IF bMove THEN
    CASE eHomeState OF
        // Wait for a rising edge
        E_MoveState.IDLING:
            IF bHomeModeEnabled AND bExecHome THEN
                bHomeDone := FALSE;
                bHomeBusy := TRUE;
                stMotionStage.bDone := FALSE;
                stDS402Drive.nDriveControl:=15;
                eHomeState :=  E_MoveState.INIT;
            END_IF
        E_MoveState.INIT:
                        stDS402Drive.nDriveControl.4:=1;
                                        eHomeState := E_MoveState.STARTED;
        E_MoveState.STARTED :
            // this is a comfirmation that routine is ongoing
            IF NOT stDS402Drive.stDriveStatus.TargetReached
                AND NOT stDS402Drive.stDriveStatus.Bit13_OpModeSpecific THEN
                bHomeBusy:=TRUE;
                bHomeDone:=FALSE;

                eHomeState:=E_MoveState.IN_PROGRESS;
            END_IF

        E_MoveState.IN_PROGRESS :

        IF bStop THEN
         stDS402Drive.nDriveControl.8 :=1;
          bHomeAborted := TRUE;
          eHomeState:=E_MoveState.INTERRUPTED;

        // Genral Motion error i.e Following error ?
        ELSIF stDS402Drive.stDriveStatus.Bit13_OpModeSpecific
                OR stDS402Drive.stDriveStatus.WarningCondition THEN
            stMotionStage.bError := TRUE;
            eHomeState:=E_MoveState.ERROR;

        // Reached
        ELSIF stDS402Drive.stDriveStatus.TargetReached
            AND stDS402Drive.stDriveStatus.Bit12_OpModeSpecific
            AND NOT stDS402Drive.stDriveStatus.Bit13_OpModeSpecific THEN
           eHomeState:=E_MoveState.DONE;
        END_IF
        E_MoveState.INTERRUPTED:
            bHomeBusy:=FALSE;
            eHomeState:=E_MoveState.IDLING;
        E_MoveState.DONE:
            bHomeBusy:=FALSE;
            bHomeDone:=TRUE;
            stMotionStage.fPosition:=0.0;

            IF (stMotionStage.nEnableMode = E_StageEnableMode.DURING_MOTION ) THEN
                stDS402Drive.nDriveControl.4:=FALSE;

            ELSE
                stDS402Drive.nDriveControl:=6;
            END_IF
            eHomeState:=E_MoveState.IDLING;
        E_MoveState.ERROR:
            bHomeDone:=FALSE;
            bHomeBusy:= FALSE;
            IF bWrongParameter THEN
                stMotionStage.sCustomErrorMessage:='Invalid motion Parameters';
                bWrongParameter := FALSE;
                stMotionStage.bError := TRUE;
            END_IF
            IF NOT stMotionStage.bError THEN
                eHomeState:=E_MoveState.IDLING;
            END_IF
    END_CASE
END_IF
END_METHOD

METHOD PUBLIC Interlock

VAR_INST
    {attribute 'hide'}
    bPositiveDirection  : BOOL;
    {attribute 'hide'}
    bNegativeDirection  : BOOL;
    {attribute 'hide'}
    ftForwardEnabled  	: F_TRIG;

    {attribute 'hide'}
    ftBackwardEnabled 	: F_TRIG;
END_VAR
// Positive or Negative direction
bPositiveDirection:=stMotionStage.bBusy AND stMotionStage.fPosDiff > 0;
bNegativeDirection:=stMotionStage.bBusy AND stMotionStage.fPosDiff < 0;

// For SmartAct MCS2 these limit are range and enstop limits. however a single bit in the status is used
// bLimOverride  : act as an override after limit was hit to allow reverse movement
stMotionStage.bLimitForwardEnable :=  bLimOverride OR NOT( bPositiveDirection AND stDS402Drive.stDriveStatus.InternalLimitActive );
stMotionStage.bLimitBackwardEnable := bLimOverride OR NOT( bNegativeDirection AND stDS402Drive.stDriveStatus.InternalLimitActive );

// use falling trigger to avoid spaming  sErrorMessage
ftForwardEnabled(CLK:=stMotionStage.bLimitForwardEnable);
ftBackwardEnabled(CLK:=stMotionStage.bLimitBackwardEnable);

IF  NOT bHomeBusy AND ftForwardEnabled.Q THEN
    // Not an error, just a warning
    stMotionStage.sCustomErrorMessage:='Cannot move past positive limit.';
    bLimOverride := TRUE;
END_IF

IF NOT bHomeBusy AND ftBackwardEnabled.Q THEN
    // Not an error, just a warning
    stMotionStage.sCustomErrorMessage:='Cannot move past Negative limit.';
    bLimOverride := TRUE;
END_IF

IF NOT stMotionStage.bError AND stMotionStage.bExecute AND NOT stMotionStage.bUserEnable THEN
    stMotionStage.bError := TRUE;
    stMotionStage.nErrorId := 1;
    stMotionStage.sCustomErrorMessage := 'Move requested, but user enable is disabled!';
END_IF

// Update all enable booleans
SetEnables();
END_METHOD

(*Switch the drive mod eof Operation
  Servo On: Profil Positioning or HOME
  Servo Off : STEP mode
*)
METHOD ModeOperation

VAR_INST
    tonSwitching : TON;
    bManualTransition: BOOL;
END_VAR
rtCSPModeOk(CLK:=( stDS402Drive.nModeOfOperationDisplay=E_DS402OpMode.CSP));
rtHomeModeEnable(CLK:=( stDS402Drive.nModeOfOperationDisplay=E_DS402OpMode.HOME));
// transition to close loop mode
IF rtCSPModeOk.Q THEN
    bHomeModeEnabled := FALSE;
    bCSPModeEnabled := TRUE;
ELSIF rtHomeModeEnable.Q THEN
    bHomeModeEnabled := TRUE;
    bCSPModeEnabled := FALSE;
    stDS402Drive.nDriveControl := 0;
END_IF

IF rtUserExec.Q AND stMotionStage.bHomeCmd THEN
    IF (stDS402Drive.nModeOfOperationDisplay<>E_DS402OpMode.HOME) THEN
        stDS402Drive.nModeOfOperation := E_DS402OpMode.HOME;
        stDS402Drive.nDriveControl := 128;
        // clear previous operational from switching away from this mode.
        bOperational := FALSE;
        bCSPModeEnabled := FALSE;
        bManualTransition := TRUE;
    ELSE
        bHomeModeEnabled := TRUE;
    END_IF
ELSIF rtUserExec.Q THEN
    IF (stDS402Drive.nModeOfOperationDisplay<>E_DS402OpMode.CSP) THEN
        stDS402Drive.nModeOfOperation := E_DS402OpMode.CSP;
        stDS402Drive.nDriveControl := 128;
        bHomeModeEnabled := FALSE;
        bManualTransition := FALSE;
    ELSE
        bCSPModeEnabled := TRUE;
    END_IF
END_IF

bDS402ManualEnabled :=bHomeModeEnabled;
(*Handle correct startup procedure for manual move*)
StateMachine(Enable:=1);
END_METHOD

METHOD PUBLIC  MoveAbsolute

fbMcMoveAbsolute(
    Axis := stMotionStage.Axis,
    Execute := bCommandMoveAbsolute,
    Position := stMotionStage.fPosition,
    Velocity := stMotionStage.fVelocity,
    Acceleration := stMotionStage.fAcceleration,
    Deceleration := stMotionStage.fDeceleration,
    BufferMode := eBufferMode,
);
END_METHOD

METHOD PersistParameters
VAR_INPUT
    Enable	: BOOL;
END_VAR

VAR_INST
    {attribute 'hide'}
    bEncError			: BOOL;

    {attribute 'hide'}
    bRestoreWaitRetry	: BOOL;
END_VAR
// Save Encoder position
// needs some pre-conditions to use persistent storage
IF Enable THEN
    // Check ST_MotionStage for an encoder error (range 0x44nn)
    bEncError:= stMotionStage.Axis.Status.Error AND  ( stMotionStage.Axis.Status.ErrorID  >= 16#4400  AND stMotionStage.Axis.Status.ErrorID <= 16#44FF );
    // Do not save if we're currently loading or if there is an encoder error
    IF NOT bRestoreLoad AND NOT bEncError AND NOT bRestoreWaitRetry THEN
        fSavedPosition := stMotionStage.Axis.NcToPlc.ActPos;
        // This persistent variable lets us check if anything was saved
        // It will be TRUE at startup if we have saved values
        bSaved := TRUE;
        (*
            use this with a timer of a change threshold on the fActPosition
            to trigger a save from this PLC program. otherwise this will be a spamming
            persistence, filling up the disk.
        *)
        //iPersistentDataStorage.TriggerWriteOfPersistentData := bSaveEnabled;
    END_IF
END_IF
END_METHOD

{attribute 'call_after_init'}
(*	eModule: Mandatory must be unique for each MCS2 axis
    clears startup errors or warnings. the process is completed at run time
    SDO update of Drive and open Loop parameter Indexes based on module number
*)
METHOD PostInit
VAR_INPUT
END_VAR
(* SDO update of Drive and open Loop parameter Indexes based on module number*)
nChanErrorCodeIdx	:= nErrorCodeBase		+ ((eModule-1) * nChanOfsBase);
nChanSoftLimitIdx	:= nChanSoftLimitBase 	+ ((eModule-1) * nChanOfsBase);
bInit := TRUE;
END_METHOD

METHOD Power : BOOL
fbMcPower(
    Axis := stMotionStage.Axis,
    Enable := stMotionStage.bAllEnable AND bCSPModeEnabled,
    Enable_Positive := stMotionStage.bAllForwardEnable,
    Enable_Negative := stMotionStage.bAllBackwardEnable,
    Override := 100.0,
    BufferMode := eBufferMode );
END_METHOD

(* Read Drive error codes after a motion or fault condition occured *)
METHOD ReadDriveCodes : BOOL
VAR_INST
    {attribute 'hide'}
    fbErrorRead			: FB_EcCoESdoRead;
    {attribute 'hide'}
    nPiezoErrorCode   	: UDINT;
    {attribute 'hide'}
    fbLogError  		: FB_LogMotionError;
    {attribute 'hide'}
    ftErrorReadDone  	: F_TRIG;
END_VAR
fbErrorRead( sNetId:= THIS^.stMotionStage.stAxisParameters.sAmsNetId,
             nSlaveAddr:=stDS402Drive.nSlaveAddr,
             nIndex:=nChanErrorCodeIdx,
             nSubIndex :=nSubIndex,
             pDstBuf:= ADR(nPiezoErrorCode),
             cbBufLen:=SIZEOF(nPiezoErrorCode),
             bExecute:= stMotionStage.bError );

ftErrorReadDone(CLK:=fbErrorRead.bBusy);
IF ftErrorReadDone.Q THEN
    IF 	NOT fbErrorRead.bError AND nPiezoErrorCode <> 0 THEN
        stMotionStage.nErrorId := nPiezoErrorCode;
    END_IF
    stMotionStage.sErrorMessage := F_MotionErrorCodeLookup(nErrorId:=stMotionStage.nErrorId);
    fbLogError( stMotionStage:=stMotionStage, bEnable:=stMotionStage.bError);
END_IF
END_METHOD

METHOD Reset : BOOL
fbMcReset(
    Axis := stMotionStage.Axis,
    Execute := bLocalReset AND bCSPModeEnabled
);

IF fbMcReset.Done OR fbMcReset.Error THEN
    bLocalReset := FALSE;
END_IF
END_METHOD

METHOD RestoreMotionParams
VAR_INPUT
    Enable	: BOOL;
END_VAR

VAR_INST
    {attribute 'hide'}
    fbSetPos			: MC_SetPosition;
    {attribute 'hide'}
    bLoad				: BOOL;
    {attribute 'hide'}
    bRestoreDone 		: BOOL;
    {attribute 'hide'}
    bRestoreInit		: BOOL;
    {attribute 'hide'}
    bRestoreWaitRetry	: BOOL;
    {attribute 'hide'}
    nMaxRetries			: UINT := 10;
    {attribute 'hide'}
    nCurrTries			: UINT := 0;
    {attribute 'hide'}
    nLatchError			: UDINT;
END_VAR
IF Enable THEN
    // Trigger a load if anything was saved at all
    IF NOT bRestoreInit THEN
        bRestoreInit := TRUE;
        bRestoreLoad S= bSaved;
        fbSetPos.Options.ClearPositionLag := TRUE;
    END_IF

    // Set our position if bRestoreLoad is true
    fbSetPos( Axis:=stMotionStage.Axis, Execute:=bRestoreLoad, Position:=fSavedPosition);

    // Only load once, at startup
    bRestoreLoad R= fbSetPos.Done OR fbSetPos.Error;

    IF fbSetPos.Error THEN
        // Keep the error latched, it can disappear if Execute is set to FALSE
        nLatchError := fbSetPos.ErrorID;
        nCurrTries := nCurrTries + 1;
        IF nCurrTries >= nMaxRetries THEN
        // Alert the user that something has gone wrong
        stMotionStage.bError := TRUE;
        stMotionStage.nErrorId := nLatchError;
        stMotionStage.sCustomErrorMessage := 'Error loading previously saved position.';
        ELSE
            // Reset the FB for the next retry
            fbSetPos( Axis:=stMotionStage.Axis, Execute:=bRestoreLoad, Position:=fSavedPosition);
            // Try again
            bRestoreWaitRetry := TRUE;
        END_IF
    ELSE
        IF NOT bRestoreDone THEN
            stMotionStage.fPosition := fSavedPosition;
        END_IF
        bRestoreDone := TRUE;
    END_IF

    tonRestoreRetry( IN := bRestoreWaitRetry, PT := T#100MS);
    bRestoreLoad S= tonRestoreRetry.Q;
    bRestoreWaitRetry R= tonRestoreRetry.Q;
END_IF
END_METHOD

METHOD ScaleDriveParams
nSoftLimMax := LREAL_TO_DINT((stMotionStage.stAxisParameters.fEncSoftEndMax / MAX(stMotionStage.stAxisParameters.fEncScaleFactorInternal, fScalingFactor)));
nSoftLimMin := LREAL_TO_DINT((stMotionStage.stAxisParameters.fEncSoftEndMin / MAX(stMotionStage.stAxisParameters.fEncScaleFactorInternal, fScalingFactor)));
END_METHOD

METHOD ScaleEncRawValue
VAR_INPUT
  //  bEnable: BOOL;
END_VAR
(* SmartACT: The encoder count from the Piezo drive is not a raw count from the embeded actuator device
   we get a calibrated nm value. thus the use of abs() since this value is signed.
   PI: to be discovered *)
IF stMotionStage.nRawEncoderDINT <> 0 THEN
    stMotionStage.nEncoderCount:=DINT_TO_UDINT(ABS(stMotionStage.nRawEncoderDINT));
ELSE
    stMotionStage.nEncoderCount:=0;
END_IF

// calibrated encoder readback
fMeasuredPos:=stMotionStage.Axis.NcToPlc.ActPos;
fMeasuredVelo :=stMotionStage.Axis.NcToPlc.ActVelo;
fMeasuredAcc := stMotionStage.Axis.NcToPlc.ActAcc;
stMotionStage.fPosDiff:=stMotionStage.Axis.NcToPlc.PosDiff;
END_METHOD

METHOD SetEnables
VAR_INPUT
END_VAR
stMotionStage.bAllForwardEnable:=stMotionStage.bLimitForwardEnable AND (stMotionStage.bGantryForwardEnable OR NOT stMotionStage.bGantryAxis) AND stMotionStage.stEPSForwardEnable.bEPS_OK;
stMotionStage.bAllBackwardEnable:=stMotionStage.bLimitBackwardEnable AND (stMotionStage.bGantryBackwardEnable OR NOT stMotionStage.bGantryAxis) AND stMotionStage.stEPSBackwardEnable.bEPS_OK;

stMotionStage.bAllEnable:=stMotionStage.bEnable AND stMotionStage.bHardwareEnable AND stMotionStage.stEPSPowerEnable.bEPS_OK;
stMotionStage.bAllEnable R= NOT stMotionStage.bUserEnable;
END_METHOD

METHOD StateMachine
VAR_INPUT
    Enable : BOOL;
END_VAR

VAR_INST
    rtFault: R_TRIG;
    {attribute 'hide'}
    bFault				: BOOL;
END_VAR
rtFault(CLK:=bFault);
(*switch on disable*)
IF NOT stDS402Drive.stDriveStatus.ReadyToSwitchOn
    AND NOT stDS402Drive.stDriveStatus.SwitchedOn
    AND NOT stDS402Drive.stDriveStatus.OperationEnabled
    AND NOT stDS402Drive.stDriveStatus.Fault
    AND stDS402Drive.stDriveStatus.VoltageEnabled
    AND NOT stDS402Drive.stDriveStatus.QuickStopActive
    AND  stDS402Drive.stDriveStatus.SwitchOnDisabled THEN
        bOperational := FALSE;
        IF bDS402ManualEnabled AND NOT bStop  THEN
            THIS^.stDS402Drive.nDriveControl := 6;
        END_IF
(*Ready to switch*)
ELSIF stDS402Drive.stDriveStatus.ReadyToSwitchOn
    AND NOT stDS402Drive.stDriveStatus.SwitchedOn
    AND NOT stDS402Drive.stDriveStatus.OperationEnabled
    AND NOT stDS402Drive.stDriveStatus.Fault
    AND stDS402Drive.stDriveStatus.VoltageEnabled
    AND stDS402Drive.stDriveStatus.QuickStopActive
    AND NOT stDS402Drive.stDriveStatus.SwitchOnDisabled THEN
        bFault := FALSE;
        bOperational := FALSE;
        IF bDS402ManualEnabled AND NOT bStop  THEN
            THIS^.stDS402Drive.nDriveControl := 7;
        END_IF
(*Switch on*)
ELSIF stDS402Drive.stDriveStatus.ReadyToSwitchOn
    AND  stDS402Drive.stDriveStatus.SwitchedOn
    AND NOT stDS402Drive.stDriveStatus.OperationEnabled
    AND NOT stDS402Drive.stDriveStatus.Fault
    AND stDS402Drive.stDriveStatus.VoltageEnabled
    AND stDS402Drive.stDriveStatus.QuickStopActive
    AND NOT stDS402Drive.stDriveStatus.SwitchOnDisabled THEN
        bOperational := FALSE;
        IF bDS402ManualEnabled AND NOT bStop  THEN
            THIS^.stDS402Drive.nDriveControl := 15;
        END_IF
(*Operation enbaled*)
ELSIF stDS402Drive.stDriveStatus.ReadyToSwitchOn
    AND stDS402Drive.stDriveStatus.SwitchedOn
    AND stDS402Drive.stDriveStatus.OperationEnabled
    AND NOT stDS402Drive.stDriveStatus.Fault
    AND stDS402Drive.stDriveStatus.VoltageEnabled
    AND stDS402Drive.stDriveStatus.QuickStopActive
    AND NOT stDS402Drive.stDriveStatus.SwitchOnDisabled THEN
        THIS^.bOperational := TRUE;
(*Fault*)
ELSIF  NOT stDS402Drive.stDriveStatus.ReadyToSwitchOn
    AND NOT stDS402Drive.stDriveStatus.SwitchedOn
    AND NOT stDS402Drive.stDriveStatus.OperationEnabled
    AND stDS402Drive.stDriveStatus.Fault
    AND stDS402Drive.stDriveStatus.VoltageEnabled
    AND NOT stDS402Drive.stDriveStatus.QuickStopActive
    AND NOT stDS402Drive.stDriveStatus.SwitchOnDisabled THEN
        bOperational := FALSE;
        bFault := TRUE;

ELSE
    bFault := FALSE;
    bOperational := FALSE;
END_IF

// wait for parameter init done at startup to read potential error from drive
stMotionStage.bError := bFault AND stMotionStage.bAxisParamsInit;
END_METHOD

(*	Drive parameters update
    Mirror NC axis parameters configurations to those of MCS2 drive
    1- Following error
    2- Home Speeds
    3- Home Acceleration
    4- SoftLimits
*)
METHOD UpdateDriveMonitoringParams
VAR_INPUT
    Enable : BOOL;
END_VAR

VAR_INST
    {attribute 'hide'}
    fbSetFErrorWin		: FB_EcCoESdoWrite;
    {attribute 'hide'}
    fbSetSoftLimMin		: FB_EcCoESdoWrite;
    {attribute 'hide'}
    fbSetSoftLimMax		: FB_EcCoESdoWrite;
    {attribute 'hide'}
    fbSetHomeOffs 		: FB_EcCoESdoWrite;
    {attribute 'hide'}
    fbSetHomeVeloFast 	: FB_EcCoESdoWrite;
    {attribute 'hide'}
    fbSetHomeVeloSlow 	: FB_EcCoESdoWrite;
    {attribute 'hide'}
    fbSetHomeAcc		: FB_EcCoESdoWrite;
    {attribute 'hide'}
    nRecentSoftLimMax 	: LINT;
    {attribute 'hide'}
    nRecentSoftLimMin 	: LINT;
    {attribute 'hide'}
    nRecentHomeVeloFast : UDINT;
    {attribute 'hide'}
    nRecentHomeVeloSlow : UDINT;
    {attribute 'hide'}
    nRecentHomeAcc 		: UDINT;
    {attribute 'hide'}
    nRecentFErrWin		: DINT;
    {attribute 'hide'}
    nRecentHomeOffset 	: DINT;
    {attribute 'hide'}
    nHomeOffs			: DINT;
    {attribute 'hide'}
    ftFErrWinSetDone	: F_TRIG;

    {attribute 'hide'}
    ftSoftLimMaxSetDone	: F_TRIG;
    {attribute 'hide'}
    ftSoftLimMinSetDone	: F_TRIG;
    {attribute 'hide'}
    ftHomeVeloFastSetDone: F_TRIG;
    {attribute 'hide'}
    ftHomeAccSetDone	: F_TRIG;
    {attribute 'hide'}
    ftHomeOffsSetDone	: F_TRIG;
    {attribute 'hide'}
    ftHomeVeloSlowSetDone: F_TRIG;
END_VAR
IF Enable THEN

    (*	Drive parameters update
        Mirror NC axis parameters configurations to those of MCS2 drive
        1- Following error.
        2- SoftLimits
        3-Position Range
    *)
  // add some safety here for  0 div.
  ScaleDriveParams();

  fbSetSoftLimMin(
    sNetId     := THIS^.stMotionStage.stAxisParameters.sAmsNetId,
    nSlaveAddr := stDS402Drive.nSlaveAddr,
    nIndex     := nChanSoftLimitIdx,
    nSubIndex  := 1,
    pSrcBuf    := ADR(nSoftLimMin),
    cbBufLen   := SIZEOF(nSoftLimMin),
    bExecute   := NOT stMotionStage.bBusy AND (nSoftLimMin <> nRecentSoftLimMin)
  );
  fbSetSoftLimMax(
    sNetId     := THIS^.stMotionStage.stAxisParameters.sAmsNetId,
    nSlaveAddr := stDS402Drive.nSlaveAddr,
    nIndex     := nChanSoftLimitIdx,
    nSubIndex  := 2,
    pSrcBuf    := ADR(nSoftLimMax),
    cbBufLen   := SIZEOF(nSoftLimMax),
    bExecute   := NOT stMotionStage.bBusy AND (nSoftLimMax <> nRecentSoftLimMax)
    );

  ftSoftLimMaxSetDone(CLK:=fbSetSoftLimMax.bBusy);
  ftSoftLimMinSetDone(CLK:=fbSetSoftLimMin.bBusy);

    IF ftSoftLimMaxSetDone.Q OR ftSoftLimMinSetDone.Q  THEN
        IF fbSetSoftLimMin.bError THEN
           stMotionStage.bError := fbSetSoftLimMin.bError;
           stMotionStage.nErrorId := fbSetSoftLimMin.nErrId;
        ELSIF fbSetSoftLimMax.bError THEN
           stMotionStage.bError := fbSetSoftLimMax.bError;
           stMotionStage.nErrorId := fbSetSoftLimMax.nErrId;
        ELSE
           nRecentSoftLimMax := nSoftLimMax;
           nRecentSoftLimMin := nSoftLimMin;
        END_IF
        fbSetSoftLimMin.bExecute := FALSE;
        fbSetSoftLimMax.bExecute := FALSE;
    END_IF
END_IF
END_METHOD

METHOD UpdateEpicsStatus
VAR_INPUT
END_VAR
//////////////////////////////////////////////////////////////////
// Transfer NC parameter status to EPICS
//////////////////////////////////////////////////////////////////
stMotionStage.stAxisStatus.bEnable:=stMotionStage.bAllEnable;
stMotionStage.stAxisStatus.bEnabled:=stMotionStage.bEnableDone; // account for PowerEnable from power block
stMotionStage.stAxisStatus.bError:=stMotionStage.bError;
stMotionStage.stAxisStatus.bHomeSensor:=stMotionStage.bHome;
stMotionStage.stAxisStatus.bLimitBwd:=stMotionStage.bAllBackwardEnable;
stMotionStage.stAxisStatus.bLimitFwd:=stMotionStage.bAllForwardEnable;
stMotionStage.stAxisStatus.bReset:=stMotionStage.bReset;
stMotionStage.stAxisStatus.fAcceleration:=fMeasuredAcc;
stMotionStage.stAxisStatus.fActDiff:=stMotionStage.fPosDiff;
stMotionStage.stAxisStatus.fActPosition:=fMeasuredPos;
stMotionStage.stAxisStatus.fActVelocity:=fMeasuredVelo;
stMotionStage.stAxisStatus.fDeceleration:=fMeasuredAcc;
stMotionStage.stAxisStatus.fOverride:=THIS^.fbMcPower.Override;
stMotionStage.stAxisStatus.fPosition:=stMotionStage.fPosition;
stMotionStage.stAxisStatus.fVelocity:=stMotionStage.fVelocity;
stMotionStage.stAxisStatus.nCmdData:=INT_TO_UINT(stMotionStage.nCmdData);  //Or nCmdDataLocal
stMotionStage.stAxisStatus.nCommand:=INT_TO_UINT(stMotionStage.nCommand);  //Or nCommandLocal
stMotionStage.stAxisStatus.nErrorId:=stMotionStage.nErrorId;
stMotionStage.stAxisStatus.bBusy:=stMotionStage.bBusy;
stMotionStage.stAxisStatus.bHomed:=stMotionStage.bHomed;
stMotionStage.stAxisStatus.bExecute:=bLocalExec;
stMotionStage.stAxisStatus.nCommand:=3; // If this is not 3, the IOC stops updating positions during homing
END_METHOD

METHOD WriteParameterNC
VAR_INPUT
    Execute:BOOL;
    ParameterNumber : MC_AxisParameter;
    ParameterValue	: LREAL;
END_VAR
(*Do not change a moving axis parameter*)
fbMcWriteParameter(	Axis:=stMotionStage.Axis,
                    Execute:=(Execute AND stMotionStage.Axis.Status.NotMoving),
                    ParameterNumber:=ParameterNumber,
                    Value:=ParameterValue
                  );

// Reset execute after when done successfull or after abort reset
// this way the done and error condition is latched till next move or global reset.
END_METHOD

END_FUNCTION_BLOCK

// ---- POUs/Motion/DS402/MCS2/FB_MCS2Calibrate.TcPOU
FUNCTION_BLOCK FB_MCS2Calibrate
VAR_INPUT
    bExecute : BOOL;
END_VAR
VAR_IN_OUT
    stDS402Drive         : ST_DS402Drive;
    stMotionStage        : ST_MotionStage;
END_VAR

VAR_OUTPUT
    bCalibrateMoveBusy        : BOOL;
    bCalibrateMoveDone        : BOOL;
    bCalibrateMoveAborted     : BOOL;
END_VAR
VAR
    eStepState	: E_MoveState := E_MoveState.IDLING;
    {attribute 'hide'}
    bReset :  BOOL;
    {attribute 'hide'}
    bHalt : BOOL;
    {attribute 'hide'}
    tonSettlingTime     : TON;
    {attribute 'hide'}
    rtCalibrateMove: R_TRIG;
END_VAR

IF NOT __ISVALIDREF(stDS402Drive)
    OR NOT __ISVALIDREF(stMotionStage) THEN
   RETURN;
END_IF

rtCalibrateMove(CLK := bExecute);

CASE eStepState OF

    E_MoveState.IDLING:
        IF rtCalibrateMove.Q THEN
            bCalibrateMoveBusy := TRUE;
            bCalibrateMoveDone := FALSE;
            // Set bits 0-3 for calibration enable
            stDS402Drive.nDriveControl.3 := TRUE;
            eStepState := E_MoveState.INIT;
        END_IF

    E_MoveState.INIT:
        // Always run the routine, even when the drive reports Calibration Attained
        // (Bit12): a Safe-Direction change invalidates the stored calibration while
        // leaving Bit12 set, so re-calibration must not be skipped.
        IF stMotionStage.bError THEN
            eStepState := E_MoveState.ERROR;
        ELSE
            stDS402Drive.nDriveControl.4 := TRUE;
            tonSettlingTime.IN:=TRUE;
            eStepState := E_MoveState.IN_PROGRESS;
        END_IF

    E_MoveState.IN_PROGRESS:
        IF bHalt OR bReset THEN
            bCalibrateMoveAborted := TRUE;
            eStepState := E_MoveState.INTERRUPTED;
        ELSIF stDS402Drive.stDriveStatus.Bit13_OpModeSpecific THEN
            stMotionStage.bError := TRUE;
            eStepState := E_MoveState.ERROR;
        ELSE
            IF tonSettlingTime.Q AND stDS402Drive.stDriveStatus.TargetReached
              AND stDS402Drive.stDriveStatus.Bit12_OpModeSpecific THEN
                eStepState := E_MoveState.REACHED;
            END_IF
        END_IF

    E_MoveState.INTERRUPTED:
        stDS402Drive.nDriveControl.4 := FALSE;
        bCalibrateMoveBusy := FALSE;
        eStepState := E_MoveState.IDLING;

    E_MoveState.REACHED:
        bCalibrateMoveBusy := FALSE;
        bCalibrateMoveDone := TRUE;
        stDS402Drive.nDriveControl.4 := FALSE;
        eStepState := E_MoveState.DONE;
    E_MoveState.DONE:
        IF stMotionStage.bDone THEN
            eStepState := E_MoveState.IDLING;
        END_IF
    E_MoveState.ERROR:
        bCalibrateMoveBusy := FALSE;
        IF NOT stMotionStage.bError THEN
            eStepState := E_MoveState.IDLING;
        END_IF

END_CASE

tonSettlingTime(PT:=T#80MS);
bHalt := FALSE;
bReset := FALSE;

METHOD Halt : BOOL
VAR_INPUT
END_VAR
THIS^.bHalt := TRUE;
END_METHOD

METHOD Reset : BOOL
VAR_INPUT
END_VAR
THIS^.bReset := TRUE;
END_METHOD

END_FUNCTION_BLOCK

// ---- POUs/Motion/DS402/MCS2/FB_MCS2Home.TcPOU
FUNCTION_BLOCK FB_MCS2Home
VAR_INPUT
    bExecute : BOOL;
END_VAR
VAR_IN_OUT
    stDS402Drive         : ST_DS402Drive;
    stMotionStage        : ST_MotionStage;
END_VAR

VAR_OUTPUT
    bHomeMoveBusy        : BOOL;
    bHomeMoveDone        : BOOL;
    bHomeMoveAborted     : BOOL;
END_VAR
VAR
    eStepState           : E_MoveState := E_MoveState.IDLING;
    {attribute 'hide'}
    bReset :  BOOL;
    {attribute 'hide'}
    bHalt : BOOL;
    {attribute 'hide'}
    tonSettlingTime     : TON;
    {attribute 'hide'}
    rtHomeMove               : R_TRIG;
    fbSetPos: MC_SetPosition;
END_VAR

IF NOT __ISVALIDREF(stDS402Drive)
    OR NOT __ISVALIDREF(stMotionStage) THEN
   RETURN;
END_IF

rtHomeMove(CLK := bExecute);

CASE eStepState OF
    E_MoveState.IDLING:
        IF rtHomeMove.Q THEN
            bHomeMoveBusy := TRUE;
            bHomeMoveDone := FALSE;
            bHomeMoveAborted := FALSE;
            stMotionStage.bDone := FALSE;
            fbSetPos.Options.ClearPositionLag := TRUE;
            tonSettlingTime.IN:=FALSE;
            stDS402Drive.nDriveControl.3 := TRUE;
            eStepState := E_MoveState.INIT;
        END_IF

    E_MoveState.INIT:
        IF stMotionStage.bError THEN
            eStepState := E_MoveState.ERROR;
        ELSE
            // Always run the full homing sequence, even when the drive already
            // reports Homing Attained (Bit12). These stick-slip stages use an
            // incremental encoder, so re-referencing to the end stop is the only
            // way to clear an undetected lost-count / slip drift. Required for
            // slit blade re-homing without a power cycle.
            stDS402Drive.nDriveControl.4 := TRUE;
            tonSettlingTime.IN:=TRUE;
            eStepState := E_MoveState.STARTED;
        END_IF

    E_MoveState.STARTED:
        IF NOT stDS402Drive.stDriveStatus.TargetReached
           AND NOT stDS402Drive.stDriveStatus.Bit13_OpModeSpecific THEN
            eStepState := E_MoveState.IN_PROGRESS;
        END_IF

    E_MoveState.IN_PROGRESS:
        IF bHalt THEN
            bHomeMoveAborted := TRUE;
            eStepState := E_MoveState.INTERRUPTED;
        ELSIF stDS402Drive.stDriveStatus.Bit13_OpModeSpecific
           OR stDS402Drive.stDriveStatus.WarningCondition THEN
            stMotionStage.bError := TRUE;
            eStepState := E_MoveState.ERROR;
        ELSIF tonSettlingTime.Q AND stDS402Drive.stDriveStatus.TargetReached
           AND stDS402Drive.stDriveStatus.Bit12_OpModeSpecific
           AND NOT stDS402Drive.stDriveStatus.Bit13_OpModeSpecific THEN
            eStepState := E_MoveState.DONE;
        END_IF

    E_MoveState.INTERRUPTED:
        stDS402Drive.nDriveControl.4 := FALSE;
        bHomeMoveBusy := FALSE;
        eStepState := E_MoveState.IDLING;

    E_MoveState.DONE:
        // Clear the homing Run bit and sync the NC to the drive readback (raw
        // count * scale + offset). Wait for MC_SetPosition to finish so the lag
        // built up during the drive-side move is cleared before homing reports
        // done. The caller re-enables position-lag monitoring and returns to CSP
        // on that done edge, so reporting early trips a following error.
        stDS402Drive.nDriveControl.4 := FALSE;
        fbSetPos(
            Axis := stMotionStage.Axis,
            Execute := TRUE,
            Position := stMotionStage.nEncoderCount
                        * stMotionStage.stAxisParameters.fEncScaleFactorInternal
                        + stMotionStage.stAxisParameters.fEncOffset
        );
        IF fbSetPos.Done THEN
            fbSetPos(Axis := stMotionStage.Axis, Execute := FALSE);
            bHomeMoveBusy := FALSE;
            bHomeMoveDone := TRUE;
            eStepState := E_MoveState.IDLING;
        ELSIF fbSetPos.Error THEN
            fbSetPos(Axis := stMotionStage.Axis, Execute := FALSE);
            bHomeMoveBusy := FALSE;
            stMotionStage.bError := TRUE;
            eStepState := E_MoveState.ERROR;
        END_IF

    E_MoveState.ERROR:
        bHomeMoveDone := FALSE;
        bHomeMoveBusy := FALSE;
        IF NOT stMotionStage.bError THEN
            eStepState := E_MoveState.IDLING;
        END_IF

END_CASE

tonSettlingTime(PT:=T#80MS);
bHalt := FALSE;
bReset := FALSE;

METHOD Halt : BOOL
VAR_INPUT
END_VAR
THIS^.bHalt := TRUE;
END_METHOD

METHOD Reset : BOOL
VAR_INPUT
END_VAR
THIS^.bReset := TRUE;
END_METHOD

END_FUNCTION_BLOCK

// ---- POUs/Motion/DS402/MCS2/FB_MCS2ReadParams.TcPOU
FUNCTION_BLOCK FB_MCS2ReadParams
VAR_IN_OUT
    stMCS2Chan1Stage : ST_MotionStage;
    stMCS2Chan2Stage : ST_MotionStage;
    stMCS2Chan3Stage : ST_MotionStage;
END_VAR
VAR
    fbReadChan1Params : FB_ReadChanParameters;
    fbReadChan2Params : FB_ReadChanParameters;
    fbReadChan3Params : FB_ReadChanParameters;
    rtExecParamsRead: R_TRIG;
    tonSDOReadTrigger: TON;
    bChanReadTrigger: BOOL;
    nReadTime : TIME  := T#2S;
END_VAR

rtExecParamsRead(CLK := (stMCS2Chan1Stage.bAxisParamsInit
                            AND stMCS2Chan2Stage.bAxisParamsInit
                            AND stMCS2Chan3Stage.bAxisParamsInit
                ));

IF rtExecParamsRead.Q THEN
    tonSDOReadTrigger(IN := TRUE);
END_IF

IF bChanReadTrigger THEN
    bChanReadTrigger := FALSE;
    tonSDOReadTrigger(IN := TRUE);
END_IF

IF tonSDOReadTrigger.Q THEN
    tonSDOReadTrigger(IN := FALSE);
    bChanReadTrigger := TRUE;
END_IF

tonSDOReadTrigger(PT := nReadTime);

END_FUNCTION_BLOCK

// ---- POUs/Motion/DS402/MCS2/FB_ReadChanParameters.TcPOU
// Two-queue serialized SDO reader for MCS2 channel parameters.
// Two independent state machines, both serializing onto the same slave but
// gated against each other so only one SDO request is outstanding at a time.
//
//   FAST queue: ChannelState only. Polled continuously at nReadTime. This is
//     the latency-sensitive path that interlocks depend on.
//
//   SLOW queue: the remaining 21 parameters (positioner type, calibration
//     options, sensor power mode, referencing options, reference type, safe
//     direction, motor load, channel type, max closed-loop frequency,
//     logical scale offset, logical scale inversion, channel temperature,
//     movement type, base unit, base resolution, distance code inverted,
//     positioner control options, actuator mode, motor load protection
//     threshold, diagnostic closed-loop frequency max and avg). Polled once
//     at boot,
//     then every nSlowReadTime (default 10 s). One read at a time. A failed
//     read logs / latches and the queue advances to the next entry.
//
// Both queues yield to each other: the fast queue will not start a new
// ChannelState read while the slow queue has one in flight, and vice versa.
// Because ChannelState reads are short (sub-100 ms) and the slow refresh
// cadence is ~10 s, ChannelState almost always wins the bus.

FUNCTION_BLOCK FB_ReadChanParameters
VAR_INPUT
    bEnable : BOOL;
END_VAR

VAR_IN_OUT
    stMotionStage       : ST_MotionStage;
    stMCS2ChanParameter : ST_MCS2ChanParameter;
    stDS402Drive        : ST_DS402Drive;
END_VAR

VAR_OUTPUT
    // TRUE once every entry in the slow queue has completed (succeeded or
    // failed) at least once. Diagnostic only -- not used to gate anything.
    bAllReadsComplete : BOOL;
    // Count of slow-queue entries that errored on their most recent attempt.
    // Cleared at the start of each slow sweep. Diagnostic only.
    nSlowReadFailures : UINT;
    // Count of fast-queue (ChannelState) reads that errored or timed out.
    // Diagnostic only -- not surfaced as a user-facing error, since polling
    // retries every cadence and a lone miss is not a fault.
    nFastReadFailures : UINT;
END_VAR

VAR

    // SDO reader instances

    // Fast queue
    fbChannelStateRead       : FB_EcCoESdoRead;
    // Event queue
    fbDriveErrCodeRead       : FB_EcCoESdoRead;
    // Slow queue
    fbMaxCloseLoopFreqRead   : FB_EcCoESdoRead;
    fbSoftLimMinRead         : FB_EcCoESdoRead;
    fbSoftLimMaxRead         : FB_EcCoESdoRead;
    fbPositionerTypeRead     : FB_EcCoESdoRead;
    fbCalibrationOptRead     : FB_EcCoESdoRead;
    fbSensorPowerModeRead    : FB_EcCoESdoRead;
    fbReferencingOptRead     : FB_EcCoESdoRead;
    fbReferenceTypeRead      : FB_EcCoESdoRead;
    fbSafeDirRead            : FB_EcCoESdoRead;
    fbMotorLoadRead          : FB_EcCoESdoRead;
    fbChannelTypeRead        : FB_EcCoESdoRead;
    fbLogicalScaleOffsetRead : FB_EcCoESdoRead;
    fbLogicalScaleInvRead    : FB_EcCoESdoRead;
    fbChannelTempRead        : FB_EcCoESdoRead;
    fbMovementTypeRead       : FB_EcCoESdoRead;
    fbBaseUnitRead           : FB_EcCoESdoRead;
    fbBaseResolutionRead     : FB_EcCoESdoRead;
    fbDistCodeInvRead        : FB_EcCoESdoRead;
    fbPositionerCtrlOptRead  : FB_EcCoESdoRead;
    fbActuatorModeRead       : FB_EcCoESdoRead;
    fbMotorLoadProtRead      : FB_EcCoESdoRead;
    // Diag closed-loop frequency is a subindexed object (0x202A:1 = max,
    // 0x202A:2 = avg); one reader per subindex.
    fbDiagClfMaxRead         : FB_EcCoESdoRead;
    fbDiagClfAvgRead         : FB_EcCoESdoRead;


    // Completion edge detectors

    ftChannelStateRead       : F_TRIG;
    ftDriveErrCodeRead       : F_TRIG;
    ftMaxCloseLoopFreqRead   : F_TRIG;
    ftSoftLimMinRead         : F_TRIG;
    ftSoftLimMaxRead         : F_TRIG;
    ftPositionerTypeRead     : F_TRIG;
    ftCalibrationOptRead     : F_TRIG;
    ftSensorPowerModeRead    : F_TRIG;
    ftReferencingOptRead     : F_TRIG;
    ftReferenceTypeRead      : F_TRIG;
    ftSafeDirRead            : F_TRIG;
    ftMotorLoadRead          : F_TRIG;
    ftChannelTypeRead        : F_TRIG;
    ftLogicalScaleOffsetRead : F_TRIG;
    ftLogicalScaleInvRead    : F_TRIG;
    ftChannelTempRead        : F_TRIG;
    ftMovementTypeRead       : F_TRIG;
    ftBaseUnitRead           : F_TRIG;
    ftBaseResolutionRead     : F_TRIG;
    ftDistCodeInvRead        : F_TRIG;
    ftPositionerCtrlOptRead  : F_TRIG;
    ftActuatorModeRead       : F_TRIG;
    ftMotorLoadProtRead      : F_TRIG;
    ftDiagClfMaxRead         : F_TRIG;
    ftDiagClfAvgRead         : F_TRIG;


    // Per-reader execute lines (driven by queue FSMs)

    bExecChannelState       : BOOL;
    bExecDriveErrCode       : BOOL;
    bExecMaxCloseLoopFreq   : BOOL;
    bExecSoftLimMin         : BOOL;
    bExecSoftLimMax         : BOOL;
    bExecPositionerType     : BOOL;
    bExecCalibrationOpt     : BOOL;
    bExecSensorPowerMode    : BOOL;
    bExecReferencingOpt     : BOOL;
    bExecReferenceType      : BOOL;
    bExecSafeDir            : BOOL;
    bExecMotorLoad          : BOOL;
    bExecChannelType        : BOOL;
    bExecLogicalScaleOffset : BOOL;
    bExecLogicalScaleInv    : BOOL;
    bExecChannelTemp        : BOOL;
    bExecMovementType       : BOOL;
    bExecBaseUnit           : BOOL;
    bExecBaseResolution     : BOOL;
    bExecDistCodeInv        : BOOL;
    bExecPositionerCtrlOpt  : BOOL;
    bExecActuatorMode       : BOOL;
    bExecMotorLoadProt      : BOOL;
    bExecDiagClfMax         : BOOL;
    bExecDiagClfAvg         : BOOL;


    // Fast queue (ChannelState)

    eFast : (
        FAST_IDLE          := 0,
        FAST_WAIT_CADENCE  := 1,
        FAST_READING       := 2
    ) := FAST_WAIT_CADENCE;
    tonFastCadence : TON;
    // Set on a fault or limit event: the drive error code reports the failed move,
    // not its cause, so the channel state bits must not be up to nReadTime stale.
    bFastReadNow : BOOL;
    // Per-read watchdog for ChannelState.
    tonFastReadTimeout : TON;
    tFastReadTimeout : TIME := T#2S;


    // Event queue (drive error code)

    // 0x603F holds the last channel error and is refreshed by the drive when the
    // Internal Limit flag is set, so it explains limit stops the NC cannot.
    eEvt : (
        EVT_IDLE    := 0,
        EVT_READING := 1
    ) := EVT_IDLE;
    rtErrEvent : R_TRIG;
    bEvtReadPending : BOOL;
    bEvtReadActive : BOOL;
    tonEvtReadTimeout : TON;
    tEvtReadTimeout : TIME := T#2S;


    // Slow queue (everything else)

    eSlow : (
        SLOW_IDLE       := 0,
        SLOW_WAIT_CADENCE := 1,
        SLOW_RUNNING    := 2
    ) := SLOW_IDLE;
    // Index into the slow-queue table. 1..NUM_SLOW; 0 = sweep complete.
    nSlowIdx : INT;
    // TRUE while a slow read is in flight (kick issued, edge not yet seen).
    bSlowReadActive : BOOL;
    tonSlowCadence : TON;
    // Per-read watchdog: if a slow read doesn't complete in tSlowReadTimeout
    // we count it as a failure, force-clear bExecute, and advance.
    tonSlowReadTimeout : TON;
    bFirstSlowSweepDone : BOOL;

    // Configurable cadences / timeouts for the slow queue.
    tSlowReadInterval : TIME := T#30S;
    tSlowReadTimeout  : TIME := T#2S;
END_VAR
VAR CONSTANT
    NUM_SLOW : INT := 23;
END_VAR

IF NOT __ISVALIDREF(stDS402Drive)
    OR NOT __ISVALIDREF(stMotionStage)
    OR NOT __ISVALIDREF(stMCS2ChanParameter) THEN
    RETURN;
END_IF

IF NOT bEnable THEN
    // Park everything off.
    bExecChannelState       := FALSE;
    bExecMaxCloseLoopFreq   := FALSE;
    bExecPositionerType     := FALSE;
    bExecCalibrationOpt     := FALSE;
    bExecSensorPowerMode    := FALSE;
    bExecReferencingOpt     := FALSE;
    bExecReferenceType      := FALSE;
    bExecSafeDir            := FALSE;
    bExecMotorLoad          := FALSE;
    bExecChannelType        := FALSE;
    bExecLogicalScaleOffset := FALSE;
    bExecLogicalScaleInv    := FALSE;
    bExecChannelTemp        := FALSE;
    bExecMovementType       := FALSE;
    bExecBaseUnit           := FALSE;
    bExecBaseResolution     := FALSE;
    bExecDistCodeInv        := FALSE;
    bExecPositionerCtrlOpt  := FALSE;
    bExecActuatorMode       := FALSE;
    bExecMotorLoadProt      := FALSE;
    bExecDiagClfMax         := FALSE;
    bExecDiagClfAvg         := FALSE;
    bExecDriveErrCode       := FALSE;
    bEvtReadPending         := FALSE;
    bEvtReadActive          := FALSE;
    bFastReadNow            := FALSE;
    eEvt                    := EVT_IDLE;
    tonEvtReadTimeout(IN := FALSE);
    tonFastCadence(IN := FALSE);
    tonSlowCadence(IN := FALSE);
    CallAllSdoReaders();
    RETURN;
END_IF

// Tick all the F_TRIGs from the previous cycle's bBusy snapshots.
ftChannelStateRead       (CLK := fbChannelStateRead.bBusy);
ftDriveErrCodeRead       (CLK := fbDriveErrCodeRead.bBusy);
ftMaxCloseLoopFreqRead   (CLK := fbMaxCloseLoopFreqRead.bBusy);
    ftSoftLimMinRead         (CLK := fbSoftLimMinRead.bBusy);
    ftSoftLimMaxRead         (CLK := fbSoftLimMaxRead.bBusy);
ftPositionerTypeRead     (CLK := fbPositionerTypeRead.bBusy);
ftCalibrationOptRead     (CLK := fbCalibrationOptRead.bBusy);
ftSensorPowerModeRead    (CLK := fbSensorPowerModeRead.bBusy);
ftReferencingOptRead     (CLK := fbReferencingOptRead.bBusy);
ftReferenceTypeRead      (CLK := fbReferenceTypeRead.bBusy);
ftSafeDirRead            (CLK := fbSafeDirRead.bBusy);
ftMotorLoadRead          (CLK := fbMotorLoadRead.bBusy);
ftChannelTypeRead        (CLK := fbChannelTypeRead.bBusy);
ftLogicalScaleOffsetRead (CLK := fbLogicalScaleOffsetRead.bBusy);
ftLogicalScaleInvRead    (CLK := fbLogicalScaleInvRead.bBusy);
ftChannelTempRead        (CLK := fbChannelTempRead.bBusy);
ftMovementTypeRead       (CLK := fbMovementTypeRead.bBusy);
ftBaseUnitRead           (CLK := fbBaseUnitRead.bBusy);
ftBaseResolutionRead     (CLK := fbBaseResolutionRead.bBusy);
ftDistCodeInvRead        (CLK := fbDistCodeInvRead.bBusy);
ftPositionerCtrlOptRead  (CLK := fbPositionerCtrlOptRead.bBusy);
ftActuatorModeRead       (CLK := fbActuatorModeRead.bBusy);
ftMotorLoadProtRead      (CLK := fbMotorLoadProtRead.bBusy);
ftDiagClfMaxRead         (CLK := fbDiagClfMaxRead.bBusy);
ftDiagClfAvgRead         (CLK := fbDiagClfAvgRead.bBusy);

// Run the two queues. Each yields to the other -- only one outstanding SDO
// at a time across the whole FB.
rtErrEvent(CLK := stMotionStage.bError OR stDS402Drive.stDriveStatus.InternalLimitActive);
IF rtErrEvent.Q THEN
    bEvtReadPending := TRUE;
    bFastReadNow    := TRUE;
END_IF

EventQueueStep();
FastQueueStep();
SlowQueueStep();

// Cyclically call every reader. bExecute lines are owned by the queues.
CallAllSdoReaders();

// Decode the raw option words into individual read-only flags.
DecodeOptions();

// Cyclic call of every SDO reader. Each FB's bExecute is owned by its queue.
METHOD PRIVATE CallAllSdoReaders
// Fast
fbChannelStateRead(
    sNetId     := stMotionStage.stAxisParameters.sAmsNetId,
    nSlaveAddr := stDS402Drive.nSlaveAddr,
    nIndex     := stMCS2ChanParameter.nChanStateIdx,
    nSubIndex  := 0,
    pDstBuf    := ADR(stMCS2ChanParameter.stChannelState.nChannelStateRaw),
    cbBufLen   := SIZEOF(stMCS2ChanParameter.stChannelState.nChannelStateRaw),
    bExecute   := bExecChannelState
);

// Event
fbDriveErrCodeRead(
    sNetId     := stMotionStage.stAxisParameters.sAmsNetId,
    nSlaveAddr := stDS402Drive.nSlaveAddr,
    nIndex     := stMCS2ChanParameter.nChanErrorCodeIdx,
    nSubIndex  := 0,
    pDstBuf    := ADR(stMCS2ChanParameter.nMCS2ErrorCode),
    cbBufLen   := SIZEOF(stMCS2ChanParameter.nMCS2ErrorCode),
    bExecute   := bExecDriveErrCode
);

// Slow
fbMaxCloseLoopFreqRead(
    sNetId     := stMotionStage.stAxisParameters.sAmsNetId,
    nSlaveAddr := stDS402Drive.nSlaveAddr,
    nIndex     := stMCS2ChanParameter.nChanMaxCloseLoopFreqIdx,
    nSubIndex  := 0,
    pDstBuf    := ADR(stMCS2ChanParameter.nMaxCloseLoopFreq),
    cbBufLen   := SIZEOF(stMCS2ChanParameter.nMaxCloseLoopFreq),
    bExecute   := bExecMaxCloseLoopFreq
);
fbSoftLimMinRead(
    sNetId     := stMotionStage.stAxisParameters.sAmsNetId,
    nSlaveAddr := stDS402Drive.nSlaveAddr,
    nIndex     := stMCS2ChanParameter.nChanSoftLimitIdx,
    nSubIndex  := 1,
    pDstBuf    := ADR(stMCS2ChanParameter.nSoftLimMin),
    cbBufLen   := SIZEOF(stMCS2ChanParameter.nSoftLimMin),
    bExecute   := bExecSoftLimMin
);
fbSoftLimMaxRead(
    sNetId     := stMotionStage.stAxisParameters.sAmsNetId,
    nSlaveAddr := stDS402Drive.nSlaveAddr,
    nIndex     := stMCS2ChanParameter.nChanSoftLimitIdx,
    nSubIndex  := 2,
    pDstBuf    := ADR(stMCS2ChanParameter.nSoftLimMax),
    cbBufLen   := SIZEOF(stMCS2ChanParameter.nSoftLimMax),
    bExecute   := bExecSoftLimMax
);
fbPositionerTypeRead(
    sNetId     := stMotionStage.stAxisParameters.sAmsNetId,
    nSlaveAddr := stDS402Drive.nSlaveAddr,
    nIndex     := stMCS2ChanParameter.nChanPositionerTypeIdx,
    nSubIndex  := 0,
    pDstBuf    := ADR(stMCS2ChanParameter.nPositionerType),
    cbBufLen   := SIZEOF(stMCS2ChanParameter.nPositionerType),
    bExecute   := bExecPositionerType
);
fbCalibrationOptRead(
    sNetId     := stMotionStage.stAxisParameters.sAmsNetId,
    nSlaveAddr := stDS402Drive.nSlaveAddr,
    nIndex     := stMCS2ChanParameter.nChanCalibrationOptIdx,
    nSubIndex  := 0,
    pDstBuf    := ADR(stMCS2ChanParameter.nCalibrationOpt),
    cbBufLen   := SIZEOF(stMCS2ChanParameter.nCalibrationOpt),
    bExecute   := bExecCalibrationOpt
);
fbSensorPowerModeRead(
    sNetId     := stMotionStage.stAxisParameters.sAmsNetId,
    nSlaveAddr := stDS402Drive.nSlaveAddr,
    nIndex     := stMCS2ChanParameter.nChanSensorPowerModeIdx,
    nSubIndex  := 0,
    pDstBuf    := ADR(stMCS2ChanParameter.nSensorPowerMode),
    cbBufLen   := SIZEOF(stMCS2ChanParameter.nSensorPowerMode),
    bExecute   := bExecSensorPowerMode
);
fbReferencingOptRead(
    sNetId     := stMotionStage.stAxisParameters.sAmsNetId,
    nSlaveAddr := stDS402Drive.nSlaveAddr,
    nIndex     := stMCS2ChanParameter.nChanReferencingOptIdx,
    nSubIndex  := 0,
    pDstBuf    := ADR(stMCS2ChanParameter.nReferencingOpt),
    cbBufLen   := SIZEOF(stMCS2ChanParameter.nReferencingOpt),
    bExecute   := bExecReferencingOpt
);
fbReferenceTypeRead(
    sNetId     := stMotionStage.stAxisParameters.sAmsNetId,
    nSlaveAddr := stDS402Drive.nSlaveAddr,
    nIndex     := stMCS2ChanParameter.nChanReferenceTypeIdx,
    nSubIndex  := 0,
    pDstBuf    := ADR(stMCS2ChanParameter.nReferenceType),
    cbBufLen   := SIZEOF(stMCS2ChanParameter.nReferenceType),
    bExecute   := bExecReferenceType
);
fbSafeDirRead(
    sNetId     := stMotionStage.stAxisParameters.sAmsNetId,
    nSlaveAddr := stDS402Drive.nSlaveAddr,
    nIndex     := stMCS2ChanParameter.nChanSafeDirIdx,
    nSubIndex  := 0,
    pDstBuf    := ADR(stMCS2ChanParameter.nSafeDir),
    cbBufLen   := SIZEOF(stMCS2ChanParameter.nSafeDir),
    bExecute   := bExecSafeDir
);
fbMotorLoadRead(
    sNetId     := stMotionStage.stAxisParameters.sAmsNetId,
    nSlaveAddr := stDS402Drive.nSlaveAddr,
    nIndex     := stMCS2ChanParameter.nChanMotorLoadIdx,
    nSubIndex  := 0,
    pDstBuf    := ADR(stMCS2ChanParameter.nMotorLoad),
    cbBufLen   := SIZEOF(stMCS2ChanParameter.nMotorLoad),
    bExecute   := bExecMotorLoad
);
fbChannelTypeRead(
    sNetId     := stMotionStage.stAxisParameters.sAmsNetId,
    nSlaveAddr := stDS402Drive.nSlaveAddr,
    nIndex     := stMCS2ChanParameter.nChannelTypeIdx,
    nSubIndex  := 0,
    pDstBuf    := ADR(stMCS2ChanParameter.nChannelType),
    cbBufLen   := SIZEOF(stMCS2ChanParameter.nChannelType),
    bExecute   := bExecChannelType
);
fbLogicalScaleOffsetRead(
    sNetId     := stMotionStage.stAxisParameters.sAmsNetId,
    nSlaveAddr := stDS402Drive.nSlaveAddr,
    nIndex     := stMCS2ChanParameter.nChanLogicalScaleOfsIdx,
    nSubIndex  := 0,
    pDstBuf    := ADR(stMCS2ChanParameter.nLogicalScaleOffset),
    cbBufLen   := SIZEOF(stMCS2ChanParameter.nLogicalScaleOffset),
    bExecute   := bExecLogicalScaleOffset
);
fbLogicalScaleInvRead(
    sNetId     := stMotionStage.stAxisParameters.sAmsNetId,
    nSlaveAddr := stDS402Drive.nSlaveAddr,
    nIndex     := stMCS2ChanParameter.nChanLogicalScaleInvIdx,
    nSubIndex  := 0,
    pDstBuf    := ADR(stMCS2ChanParameter.nLogicalScaleInv),
    cbBufLen   := SIZEOF(stMCS2ChanParameter.nLogicalScaleInv),
    bExecute   := bExecLogicalScaleInv
);
fbChannelTempRead(
    sNetId     := stMotionStage.stAxisParameters.sAmsNetId,
    nSlaveAddr := stDS402Drive.nSlaveAddr,
    nIndex     := stMCS2ChanParameter.nChanChannelTempIdx,
    nSubIndex  := 0,
    pDstBuf    := ADR(stMCS2ChanParameter.nChannelTemp),
    cbBufLen   := SIZEOF(stMCS2ChanParameter.nChannelTemp),
    bExecute   := bExecChannelTemp
);
fbMovementTypeRead(
    sNetId     := stMotionStage.stAxisParameters.sAmsNetId,
    nSlaveAddr := stDS402Drive.nSlaveAddr,
    nIndex     := stMCS2ChanParameter.nChanMovementTypeIdx,
    nSubIndex  := 0,
    pDstBuf    := ADR(stMCS2ChanParameter.nMovementType),
    cbBufLen   := SIZEOF(stMCS2ChanParameter.nMovementType),
    bExecute   := bExecMovementType
);
fbBaseUnitRead(
    sNetId     := stMotionStage.stAxisParameters.sAmsNetId,
    nSlaveAddr := stDS402Drive.nSlaveAddr,
    nIndex     := stMCS2ChanParameter.nChanBaseUnitIdx,
    nSubIndex  := 0,
    pDstBuf    := ADR(stMCS2ChanParameter.nBaseUnit),
    cbBufLen   := SIZEOF(stMCS2ChanParameter.nBaseUnit),
    bExecute   := bExecBaseUnit
);
fbBaseResolutionRead(
    sNetId     := stMotionStage.stAxisParameters.sAmsNetId,
    nSlaveAddr := stDS402Drive.nSlaveAddr,
    nIndex     := stMCS2ChanParameter.nChanBaseResolutionIdx,
    nSubIndex  := 0,
    pDstBuf    := ADR(stMCS2ChanParameter.nBaseResolution),
    cbBufLen   := SIZEOF(stMCS2ChanParameter.nBaseResolution),
    bExecute   := bExecBaseResolution
);
fbDistCodeInvRead(
    sNetId     := stMotionStage.stAxisParameters.sAmsNetId,
    nSlaveAddr := stDS402Drive.nSlaveAddr,
    nIndex     := stMCS2ChanParameter.nChanDistCodeInvIdx,
    nSubIndex  := 0,
    pDstBuf    := ADR(stMCS2ChanParameter.nDistCodeInv),
    cbBufLen   := SIZEOF(stMCS2ChanParameter.nDistCodeInv),
    bExecute   := bExecDistCodeInv
);
fbPositionerCtrlOptRead(
    sNetId     := stMotionStage.stAxisParameters.sAmsNetId,
    nSlaveAddr := stDS402Drive.nSlaveAddr,
    nIndex     := stMCS2ChanParameter.nChanPositionerCtrlOptIdx,
    nSubIndex  := 0,
    pDstBuf    := ADR(stMCS2ChanParameter.nPositionerCtrlOpt),
    cbBufLen   := SIZEOF(stMCS2ChanParameter.nPositionerCtrlOpt),
    bExecute   := bExecPositionerCtrlOpt
);
fbActuatorModeRead(
    sNetId     := stMotionStage.stAxisParameters.sAmsNetId,
    nSlaveAddr := stDS402Drive.nSlaveAddr,
    nIndex     := stMCS2ChanParameter.nChanActuatorModeIdx,
    nSubIndex  := 0,
    pDstBuf    := ADR(stMCS2ChanParameter.nActuatorMode),
    cbBufLen   := SIZEOF(stMCS2ChanParameter.nActuatorMode),
    bExecute   := bExecActuatorMode
);
fbMotorLoadProtRead(
    sNetId     := stMotionStage.stAxisParameters.sAmsNetId,
    nSlaveAddr := stDS402Drive.nSlaveAddr,
    nIndex     := stMCS2ChanParameter.nChanMotorLoadProtIdx,
    nSubIndex  := 0,
    pDstBuf    := ADR(stMCS2ChanParameter.nMotorLoadProt),
    cbBufLen   := SIZEOF(stMCS2ChanParameter.nMotorLoadProt),
    bExecute   := bExecMotorLoadProt
);
fbDiagClfMaxRead(
    sNetId     := stMotionStage.stAxisParameters.sAmsNetId,
    nSlaveAddr := stDS402Drive.nSlaveAddr,
    nIndex     := stMCS2ChanParameter.nChanDiagClfIdx,
    nSubIndex  := 1,
    pDstBuf    := ADR(stMCS2ChanParameter.nDiagClfMax),
    cbBufLen   := SIZEOF(stMCS2ChanParameter.nDiagClfMax),
    bExecute   := bExecDiagClfMax
);
fbDiagClfAvgRead(
    sNetId     := stMotionStage.stAxisParameters.sAmsNetId,
    nSlaveAddr := stDS402Drive.nSlaveAddr,
    nIndex     := stMCS2ChanParameter.nChanDiagClfIdx,
    nSubIndex  := 2,
    pDstBuf    := ADR(stMCS2ChanParameter.nDiagClfAvg),
    cbBufLen   := SIZEOF(stMCS2ChanParameter.nDiagClfAvg),
    bExecute   := bExecDiagClfAvg
);
END_METHOD

METHOD PRIVATE ClearAllSlowExecutes
bExecMaxCloseLoopFreq   := FALSE;
bExecPositionerType     := FALSE;
bExecCalibrationOpt     := FALSE;
bExecSensorPowerMode    := FALSE;
bExecReferencingOpt     := FALSE;
bExecReferenceType      := FALSE;
bExecSafeDir            := FALSE;
bExecMotorLoad          := FALSE;
bExecChannelType        := FALSE;
bExecLogicalScaleOffset := FALSE;
bExecLogicalScaleInv    := FALSE;
bExecChannelTemp        := FALSE;
bExecMovementType       := FALSE;
bExecBaseUnit           := FALSE;
bExecBaseResolution     := FALSE;
bExecDistCodeInv        := FALSE;
bExecPositionerCtrlOpt  := FALSE;
bExecActuatorMode       := FALSE;
bExecMotorLoadProt      := FALSE;
bExecDiagClfMax         := FALSE;
bExecDiagClfAvg         := FALSE;
bExecSoftLimMin         := FALSE;
bExecSoftLimMax         := FALSE;
END_METHOD

METHOD PRIVATE ClearSlowExecute
VAR_INPUT
    idx : INT;
END_VAR
CASE idx OF
    1:  bExecMaxCloseLoopFreq   := FALSE;
    2:  bExecPositionerType     := FALSE;
    3:  bExecCalibrationOpt     := FALSE;
    4:  bExecSensorPowerMode    := FALSE;
    5:  bExecReferencingOpt     := FALSE;
    6:  bExecReferenceType      := FALSE;
    7:  bExecSafeDir            := FALSE;
    8:  bExecMotorLoad          := FALSE;
    9:  bExecChannelType        := FALSE;
    10: bExecLogicalScaleOffset := FALSE;
    11: bExecLogicalScaleInv    := FALSE;
    12: bExecChannelTemp        := FALSE;
    13: bExecMovementType       := FALSE;
    14: bExecBaseUnit           := FALSE;
    15: bExecBaseResolution     := FALSE;
    16: bExecDistCodeInv        := FALSE;
    17: bExecPositionerCtrlOpt  := FALSE;
    18: bExecActuatorMode       := FALSE;
    19: bExecMotorLoadProt      := FALSE;
    20: bExecDiagClfMax         := FALSE;
    21: bExecDiagClfAvg         := FALSE;
    22: bExecSoftLimMin         := FALSE;
    23: bExecSoftLimMax         := FALSE;
END_CASE
END_METHOD

// Unpack the 32-bit raw channel state word into individual flag fields.
METHOD PRIVATE DecodeChannelState
VAR
    n : UDINT;
END_VAR
n := stMCS2ChanParameter.stChannelState.nChannelStateRaw;
stMCS2ChanParameter.stChannelState.bActivelyMoving        := (n AND 16#00000001) <> 0;
stMCS2ChanParameter.stChannelState.bClosedLoopActive      := (n AND 16#00000002) <> 0;
stMCS2ChanParameter.stChannelState.bCalibrating           := (n AND 16#00000004) <> 0;
stMCS2ChanParameter.stChannelState.bReferencing           := (n AND 16#00000008) <> 0;
stMCS2ChanParameter.stChannelState.bMoveDelayed           := (n AND 16#00000010) <> 0;
stMCS2ChanParameter.stChannelState.bSensorPresent         := (n AND 16#00000020) <> 0;
stMCS2ChanParameter.stChannelState.bIsCalibrated          := (n AND 16#00000040) <> 0;
stMCS2ChanParameter.stChannelState.bIsReferenced          := (n AND 16#00000080) <> 0;
stMCS2ChanParameter.stChannelState.bEndStopReached        := (n AND 16#00000100) <> 0;
stMCS2ChanParameter.stChannelState.bRangeLimitReached     := (n AND 16#00000200) <> 0;
stMCS2ChanParameter.stChannelState.bFollowingLimitReached := (n AND 16#00000400) <> 0;
stMCS2ChanParameter.stChannelState.bMovementFailed        := (n AND 16#00000800) <> 0;
stMCS2ChanParameter.stChannelState.bIsStreaming           := (n AND 16#00001000) <> 0;
stMCS2ChanParameter.stChannelState.bPositionerOverload    := (n AND 16#00002000) <> 0;
stMCS2ChanParameter.stChannelState.bOverTemperature       := (n AND 16#00004000) <> 0;
stMCS2ChanParameter.stChannelState.bReferenceMark         := (n AND 16#00008000) <> 0;
stMCS2ChanParameter.stChannelState.bIsPhased              := (n AND 16#00010000) <> 0;
stMCS2ChanParameter.stChannelState.bPositionerFault       := (n AND 16#00020000) <> 0;
stMCS2ChanParameter.stChannelState.bAmplifierEnabled      := (n AND 16#00040000) <> 0;
stMCS2ChanParameter.stChannelState.bInPosition            := (n AND 16#00080000) <> 0;
stMCS2ChanParameter.stChannelState.bBrakeEnabled          := (n AND 16#00100000) <> 0;

// Preserve a useful MCS2 diagnostic even if the asynchronous 0x603F read is
// delayed or unavailable. The SDO result, when available, replaces this
// inferred summary with the drive's exact code.
IF stMCS2ChanParameter.stChannelState.bRangeLimitReached THEN
    stMCS2ChanParameter.nMCS2ErrorCode := 16#8500;
ELSIF stMCS2ChanParameter.stChannelState.bEndStopReached THEN
    stMCS2ChanParameter.nMCS2ErrorCode := 16#7121;
ELSIF stMCS2ChanParameter.stChannelState.bFollowingLimitReached THEN
    stMCS2ChanParameter.nMCS2ErrorCode := 16#8611;
ELSIF stMCS2ChanParameter.stChannelState.bMovementFailed THEN
    stMCS2ChanParameter.nMCS2ErrorCode := 16#8600;
END_IF
END_METHOD

// Decode the raw Referencing Options (0x200B) and Calibration Options (0x2004)
// words read back from the drive into individual read-only flags.
METHOD PRIVATE DecodeOptions
VAR
    n : DWORD;
END_VAR
n := stMCS2ChanParameter.nReferencingOpt;
stMCS2ChanParameter.bRefStartDirBackward   := (n AND 16#00000001) <> 0;
stMCS2ChanParameter.bRefReverseDir         := (n AND 16#00000002) <> 0;
stMCS2ChanParameter.bRefAutoZero           := (n AND 16#00000004) <> 0;
stMCS2ChanParameter.bRefAbortOnEndStop     := (n AND 16#00000008) <> 0;
stMCS2ChanParameter.bRefContinueOnRefFound := (n AND 16#00000010) <> 0;
stMCS2ChanParameter.bRefStopOnRefFound     := (n AND 16#00000020) <> 0;
stMCS2ChanParameter.bRefInvalidate         := (n AND 16#01000000) <> 0;

n := stMCS2ChanParameter.nCalibrationOpt;
stMCS2ChanParameter.bCalDirBackward        := (n AND 16#00000001) <> 0;
stMCS2ChanParameter.bCalDetectDistCodeInv  := (n AND 16#00000002) <> 0;
stMCS2ChanParameter.bCalAdvSensorCorr      := (n AND 16#00000004) <> 0;
stMCS2ChanParameter.bCalLimitedTravelRange := (n AND 16#00000100) <> 0;
END_METHOD

// Event queue: one-shot read of the drive error code (0x603F) after a fault or
// internal-limit event. Highest priority, but still mutually exclusive with the
// fast and slow queues so only one SDO is outstanding on the mailbox.
METHOD PRIVATE EventQueueStep
CASE eEvt OF

    EVT_IDLE:
        bExecDriveErrCode := FALSE;
        bEvtReadActive    := FALSE;
        tonEvtReadTimeout(IN := FALSE);
        IF bEvtReadPending
           AND NOT bSlowReadActive
           AND (eFast <> FAST_READING) THEN
            bEvtReadPending   := FALSE;
            bExecDriveErrCode := TRUE;
            bEvtReadActive    := TRUE;
            eEvt              := EVT_READING;
        END_IF

    EVT_READING:
        tonEvtReadTimeout(IN := TRUE, PT := tEvtReadTimeout);
        IF ftDriveErrCodeRead.Q THEN
            // Keep an inferred or previously read code if this mailbox read
            // fails. ChannelState provides a useful cause-level fallback.
            bExecDriveErrCode := FALSE;
            bEvtReadActive    := FALSE;
            tonEvtReadTimeout(IN := FALSE);
            eEvt              := EVT_IDLE;
        ELSIF tonEvtReadTimeout.Q THEN
            // Keep the inferred or previously read code for diagnostics.
            bExecDriveErrCode := FALSE;
            bEvtReadActive    := FALSE;
            tonEvtReadTimeout(IN := FALSE);
            eEvt              := EVT_IDLE;
        END_IF

END_CASE
END_METHOD

// Fast queue: poll ChannelState at nReadTime cadence. Yields the bus to the
// slow and event queues if one of those reads is currently in flight, but does
// not back off any further -- as soon as that read completes the fast read can fire.
METHOD PRIVATE FastQueueStep
CASE eFast OF

    FAST_IDLE:
        bExecChannelState := FALSE;
        eFast             := FAST_WAIT_CADENCE;

    FAST_WAIT_CADENCE:
        bExecChannelState := FALSE;
        tonFastReadTimeout(IN := FALSE);
        // Cadence timer runs while we're waiting for our next turn.
        tonFastCadence(
            IN := stMotionStage.bAxisParamsInit,
            PT := stMCS2ChanParameter.nReadTime
        );
        // Only fire when the cadence has elapsed AND the slow queue isn't
        // currently using the mailbox.
        IF (tonFastCadence.Q OR bFastReadNow) AND NOT bSlowReadActive AND NOT bEvtReadActive THEN
            tonFastCadence(IN := FALSE);
            bFastReadNow      := FALSE;
            bExecChannelState := TRUE;
            eFast             := FAST_READING;
        END_IF

    FAST_READING:
        // Hold execute TRUE through the read. F_TRIG on bBusy falling = done.
        tonFastReadTimeout(IN := TRUE, PT := tFastReadTimeout);
        IF ftChannelStateRead.Q THEN
            IF NOT fbChannelStateRead.bError THEN
                DecodeChannelState();
            ELSE
                // Don't stop polling on a single failure, and don't surface
                // it as a user-facing error -- it retries every cadence.
                nFastReadFailures := nFastReadFailures + 1;
            END_IF
            bExecChannelState := FALSE;
            tonFastReadTimeout(IN := FALSE);
            eFast             := FAST_WAIT_CADENCE;
        ELSIF tonFastReadTimeout.Q THEN
            // Hung read -- give up and retry next cadence.
            nFastReadFailures := nFastReadFailures + 1;
            bExecChannelState := FALSE;
            tonFastReadTimeout(IN := FALSE);
            eFast             := FAST_WAIT_CADENCE;
        END_IF

END_CASE
END_METHOD

// Slow queue: sweep through 21 entries once at boot, then refresh every
// tSlowReadInterval. One entry at a time. A failed read latches a counter
// and advances -- it does not stall the sweep or affect the fast queue.
METHOD PRIVATE SlowQueueStep
CASE eSlow OF

    SLOW_IDLE:
        ClearAllSlowExecutes();
        bSlowReadActive := FALSE;
        // Begin first sweep as soon as axis params are initialized.
        IF stMotionStage.bAxisParamsInit THEN
            nSlowIdx          := 1;
            nSlowReadFailures := 0;
            eSlow             := SLOW_RUNNING;
        END_IF

    SLOW_WAIT_CADENCE:
        ClearAllSlowExecutes();
        bSlowReadActive := FALSE;
        tonSlowCadence(
            IN := stMotionStage.bAxisParamsInit,
            PT := tSlowReadInterval
        );
        IF tonSlowCadence.Q THEN
            tonSlowCadence(IN := FALSE);
            nSlowIdx          := 1;
            nSlowReadFailures := 0;
            eSlow             := SLOW_RUNNING;
        END_IF

    SLOW_RUNNING:
        // Yield: never start a new slow read while the fast queue is
        // mid-read. Existing in-flight slow reads continue.
        IF NOT bSlowReadActive AND ((eFast = FAST_READING) OR bEvtReadActive) THEN
            // Just hold; don't kick the next read yet.
            RETURN;
        END_IF

        IF NOT bSlowReadActive THEN
            // Start the read at the current index.
            StartSlowRead(nSlowIdx);
            bSlowReadActive := TRUE;
            tonSlowReadTimeout(IN := FALSE);   // reset
        ELSE
            // Arm watchdog while we wait.
            tonSlowReadTimeout(IN := TRUE, PT := tSlowReadTimeout);
            IF SlowReadEdge(nSlowIdx) THEN
                // Normal completion path.
                IF SlowReadError(nSlowIdx) THEN
                    nSlowReadFailures := nSlowReadFailures + 1;
                END_IF
                ClearSlowExecute(nSlowIdx);
                bSlowReadActive := FALSE;
                tonSlowReadTimeout(IN := FALSE);
                nSlowIdx := nSlowIdx + 1;
            ELSIF tonSlowReadTimeout.Q THEN
                // Hung read -- force-clear and advance. The reader FB will
                // see bExecute drop; whether it ever asserts an edge later
                // is its problem, not ours.
                nSlowReadFailures := nSlowReadFailures + 1;
                ClearSlowExecute(nSlowIdx);
                bSlowReadActive := FALSE;
                tonSlowReadTimeout(IN := FALSE);
                nSlowIdx := nSlowIdx + 1;
            END_IF

            IF nSlowIdx > NUM_SLOW THEN
                // Sweep done.
                bFirstSlowSweepDone := TRUE;
                bAllReadsComplete   := TRUE;
                nSlowIdx            := 0;
                eSlow               := SLOW_WAIT_CADENCE;
            END_IF
        END_IF

END_CASE
END_METHOD

// Return TRUE on the cycle the read at <idx> completes (busy->idle).
METHOD PRIVATE SlowReadEdge : BOOL
VAR_INPUT
    idx : INT;
END_VAR
CASE idx OF
    1:  SlowReadEdge := ftMaxCloseLoopFreqRead.Q;
    2:  SlowReadEdge := ftPositionerTypeRead.Q;
    3:  SlowReadEdge := ftCalibrationOptRead.Q;
    4:  SlowReadEdge := ftSensorPowerModeRead.Q;
    5:  SlowReadEdge := ftReferencingOptRead.Q;
    6:  SlowReadEdge := ftReferenceTypeRead.Q;
    7:  SlowReadEdge := ftSafeDirRead.Q;
    8:  SlowReadEdge := ftMotorLoadRead.Q;
    9:  SlowReadEdge := ftChannelTypeRead.Q;
    10: SlowReadEdge := ftLogicalScaleOffsetRead.Q;
    11: SlowReadEdge := ftLogicalScaleInvRead.Q;
    12: SlowReadEdge := ftChannelTempRead.Q;
    13: SlowReadEdge := ftMovementTypeRead.Q;
    14: SlowReadEdge := ftBaseUnitRead.Q;
    15: SlowReadEdge := ftBaseResolutionRead.Q;
    16: SlowReadEdge := ftDistCodeInvRead.Q;
    17: SlowReadEdge := ftPositionerCtrlOptRead.Q;
    18: SlowReadEdge := ftActuatorModeRead.Q;
    19: SlowReadEdge := ftMotorLoadProtRead.Q;
    20: SlowReadEdge := ftDiagClfMaxRead.Q;
    21: SlowReadEdge := ftDiagClfAvgRead.Q;
    22: SlowReadEdge := ftSoftLimMinRead.Q;
    23: SlowReadEdge := ftSoftLimMaxRead.Q;
    ELSE
        SlowReadEdge := FALSE;
END_CASE
END_METHOD

// Return the .bError flag for the read at <idx> after completion.
METHOD PRIVATE SlowReadError : BOOL
VAR_INPUT
    idx : INT;
END_VAR
CASE idx OF
    1:  SlowReadError := fbMaxCloseLoopFreqRead.bError;
    2:  SlowReadError := fbPositionerTypeRead.bError;
    3:  SlowReadError := fbCalibrationOptRead.bError;
    4:  SlowReadError := fbSensorPowerModeRead.bError;
    5:  SlowReadError := fbReferencingOptRead.bError;
    6:  SlowReadError := fbReferenceTypeRead.bError;
    7:  SlowReadError := fbSafeDirRead.bError;
    8:  SlowReadError := fbMotorLoadRead.bError;
    9:  SlowReadError := fbChannelTypeRead.bError;
    10: SlowReadError := fbLogicalScaleOffsetRead.bError;
    11: SlowReadError := fbLogicalScaleInvRead.bError;
    12: SlowReadError := fbChannelTempRead.bError;
    13: SlowReadError := fbMovementTypeRead.bError;
    14: SlowReadError := fbBaseUnitRead.bError;
    15: SlowReadError := fbBaseResolutionRead.bError;
    16: SlowReadError := fbDistCodeInvRead.bError;
    17: SlowReadError := fbPositionerCtrlOptRead.bError;
    18: SlowReadError := fbActuatorModeRead.bError;
    19: SlowReadError := fbMotorLoadProtRead.bError;
    20: SlowReadError := fbDiagClfMaxRead.bError;
    21: SlowReadError := fbDiagClfAvgRead.bError;
    22: SlowReadError := fbSoftLimMinRead.bError;
    23: SlowReadError := fbSoftLimMaxRead.bError;
    ELSE
        SlowReadError := FALSE;
END_CASE
END_METHOD

// Issue bExecute=TRUE for the slow-queue entry at the given index.
METHOD PRIVATE StartSlowRead
VAR_INPUT
    idx : INT;
END_VAR
CASE idx OF
    1:  bExecMaxCloseLoopFreq   := TRUE;
    2:  bExecPositionerType     := TRUE;
    3:  bExecCalibrationOpt     := TRUE;
    4:  bExecSensorPowerMode    := TRUE;
    5:  bExecReferencingOpt     := TRUE;
    6:  bExecReferenceType      := TRUE;
    7:  bExecSafeDir            := TRUE;
    8:  bExecMotorLoad          := TRUE;
    9:  bExecChannelType        := TRUE;
    10: bExecLogicalScaleOffset := TRUE;
    11: bExecLogicalScaleInv    := TRUE;
    12: bExecChannelTemp        := TRUE;
    13: bExecMovementType       := TRUE;
    14: bExecBaseUnit           := TRUE;
    15: bExecBaseResolution     := TRUE;
    16: bExecDistCodeInv        := TRUE;
    17: bExecPositionerCtrlOpt  := TRUE;
    18: bExecActuatorMode       := TRUE;
    19: bExecMotorLoadProt      := TRUE;
    20: bExecDiagClfMax         := TRUE;
    21: bExecDiagClfAvg         := TRUE;
    22: bExecSoftLimMin         := TRUE;
    23: bExecSoftLimMax         := TRUE;
END_CASE
END_METHOD

END_FUNCTION_BLOCK

// ---- POUs/Motion/DS402/MCS2/FB_MCS2StepMode.TcPOU
FUNCTION_BLOCK FB_MCS2StepMode
VAR_INPUT
    bExecute : BOOL;
END_VAR
VAR_IN_OUT
    stDS402Drive         : ST_DS402Drive;
    stMotionStage        : ST_MotionStage;
END_VAR

VAR_OUTPUT
    bStepMoveBusy        : BOOL;
    bStepMoveDone        : BOOL;
    bStepMoveAborted     : BOOL;
END_VAR
VAR
    eStepState           : E_MoveState := E_MoveState.IDLING;
    bReset :  BOOL;
    bHalt : BOOL;
    tonSettlingTime     : TON;
    {attribute 'hide'}
    rtStepMove               : R_TRIG;
END_VAR

IF NOT __ISVALIDREF(stDS402Drive)
    OR NOT __ISVALIDREF(stMotionStage)  THEN
   RETURN;
END_IF

rtStepMove(CLK := bExecute);

CASE eStepState OF
    E_MoveState.IDLING:
        IF rtStepMove.Q THEN
            bStepMoveBusy := TRUE;
            bStepMoveDone := FALSE;
            bStepMoveAborted := FALSE;
            tonSettlingTime.IN:=FALSE;
            stDS402Drive.nDriveControl.3 := TRUE;
            eStepState := E_MoveState.INIT;
        END_IF

    E_MoveState.INIT:
        IF stMotionStage.bError THEN
            eStepState := E_MoveState.ERROR;
        ELSE
            stDS402Drive.nDriveControl.4 := TRUE;
            tonSettlingTime.IN:=TRUE;
            eStepState := E_MoveState.IN_PROGRESS;
        END_IF

    E_MoveState.IN_PROGRESS:
        IF bHalt OR bReset THEN
            bStepMoveAborted := TRUE;
            eStepState := E_MoveState.INTERRUPTED;
        ELSIF stDS402Drive.stDriveStatus.Bit13_OpModeSpecific THEN
            stMotionStage.bError := TRUE;
            eStepState := E_MoveState.ERROR;
        ELSE
            IF tonSettlingTime.Q AND stDS402Drive.stDriveStatus.TargetReached THEN
                eStepState := E_MoveState.REACHED;
            END_IF
        END_IF

    E_MoveState.INTERRUPTED:
        stDS402Drive.nDriveControl.4 := FALSE;
        bStepMoveBusy := FALSE;
        eStepState := E_MoveState.IDLING;

    E_MoveState.REACHED:
        bStepMoveBusy := FALSE;
        bStepMoveDone := TRUE;
        stDS402Drive.nDriveControl.4 := FALSE;
        eStepState := E_MoveState.DONE;

    E_MoveState.DONE:
        IF stMotionStage.bDone THEN
            eStepState := E_MoveState.IDLING;
        END_IF

    E_MoveState.ERROR:
        bStepMoveBusy := FALSE;
        bStepMoveDone := FALSE;
        IF NOT stMotionStage.bError THEN
            eStepState := E_MoveState.IDLING;
        END_IF
END_CASE
tonSettlingTime(PT:=T#80MS);
bHalt := FALSE;
bReset := FALSE;

METHOD Halt : BOOL
VAR_INPUT
END_VAR
THIS^.bHalt := TRUE;
END_METHOD

METHOD Reset : BOOL
VAR_INPUT
END_VAR
THIS^.bReset := TRUE;
END_METHOD

END_FUNCTION_BLOCK

// ---- POUs/Motion/DS402/MCS2/FB_MotionStageMCS2.TcPOU
(*
    MCS2 Motion Stage
    Controls a stage in CSP (NC), STEP_MODE, and Homing via DS402 interface.
    - Uses overridden Position Holding timer.
    - power enable mode must be 'DURING_MOTION' for closed-loop (CSP) control.
    - Set bServo PV to true for closed-loop, clear for open-loop (step mode).
*)
{attribute 'call_after_init'}
FUNCTION_BLOCK FB_MotionStageMCS2

VAR
    {attribute 'no_copy'}
    stMotionStage		: REFERENCE TO ST_MotionStage;
    {attribute 'no_copy'}
    stChanParams       : REFERENCE TO ST_MCS2ChanParameter;
    // Hardware I/O
    {attribute 'pytmc' := 'pv:'}
    stDS402Drive		: ST_DS402Drive;

    fbDriveManager		: FB_MCS2DriveManager;
    fbReadChanParams	: FB_ReadChanParameters;
    fbStepMode 			: FB_MCS2StepMode;
    fbhome 				: FB_MCS2Home;
    fbCalibrate			: FB_MCS2Calibrate;
    fbWriteParameters 	: FB_WriteChanParameters;
    fbReadDriveCodes 	: FB_ReadDriveCodes;

    {attribute 'hide'}
    eModule                 : E_Module;
    {attribute 'hide'}
    eDoneCause              : E_MoveDoneCause := E_MoveDoneCause.Unknown;
    {attribute 'hide'}
    fbMcPower               : MC_Power;
    {attribute 'hide'}
    fbMcMoveAbsolute        : MC_MoveAbsolute;
    {attribute 'hide'}
    fbMcHalt                : MC_Halt;
    {attribute 'hide'}
    fbMcReset               : MC_Reset;
    {attribute 'hide'}
    fbMcWriteParameter      : MC_WriteParameter;
    {attribute 'hide'}
    fbMcReadParams          : MC_ReadParameterSet;
    {attribute 'hide'}
    fParameterValue : LREAL;
    fMeasuredPos: LREAL;
    fMeasuredVelo: LREAL;
    fMeasuredAcc: LREAL;
    bLastHoltTimeOut : BOOL;
    bRestoreWaitRetry   : BOOL;
    {attribute 'hide'}
    bEnPosLag               : BOOL;
    {attribute 'hide'}
    bWrongParameter         : BOOL;
    {attribute 'hide'}
    bExecMove               : BOOL;
    {attribute 'hide'}
    bExecHome               : BOOL;
    {attribute 'hide'}
    bNewMoveReq             : BOOL;
    {attribute 'hide'}
    bPrepareDisable         : BOOL;
    {attribute 'hide'}
    bHalt                   : BOOL;
    {attribute 'hide'}
    bLimOverride            : BOOL;
    {attribute 'hide'}
    bPositionHold           : BOOL;
    {attribute 'hide'}
    bLocalExec              : BOOL;
    {attribute 'hide'}
    bSystemInit             : BOOL;
    {attribute 'hide'}
    bRestoreLoad             : BOOL;
    {attribute 'hide'}
    bExecParamRead          : BOOL;

    {attribute 'hide'}
    bRecentEnPosLagStatus    : BOOL;

    {attribute 'hide'}
    bLagClearPending         : BOOL;
    {attribute 'hide'}
    tonLagClearTimeout       : TON;
    {attribute 'hide'}
    rtMcWriteDone            : R_TRIG;

    {attribute 'hide'}
    bReset                   : BOOL;
    bFault : BOOL := FALSE;
    {attribute 'hide'}
    nCmdDataLocal            : INT;
    tonHoldTime              : TON;
    {attribute 'hide'}
    NCParamsTimer            : TON;
    {attribute 'hide'}
    tonRestoreRetry          : TON;
    {attribute 'hide'}
    rtExec                   : R_TRIG;
    {attribute 'hide'}
    rtMoveCmdShortcut        : R_TRIG;
    {attribute 'hide'}
    rtHomeCmdShortcut        : R_TRIG;
    {attribute 'hide'}
    rtEnableMode             : R_TRIG;
    {attribute 'hide'}
    rtUserExec               : R_TRIG;
    {attribute 'hide'}
    rtMoveDone               : R_TRIG;
    {attribute 'hide'}
    rtNewMoveReq             : R_TRIG;
    {attribute 'hide'}
    ftExec                   : F_TRIG;
    rtHaltEdge : R_TRIG;
    {attribute 'hide'}
    rtStepCmdShortcut		 : R_TRIG;
    {attribute 'hide'}
    rtStepFwdCmdShortcut	 : R_TRIG;
    {attribute 'hide'}
    rtStepRevCmdShortcut	 : R_TRIG;
    {attribute 'hide'}
    rtCalibrateCmdShortcut	 : R_TRIG;
    {attribute 'hide'}
    tSDOOpsTimer 			 : TON;
    {attribute 'hide'}
    bParamsEnable			 : BOOL;
    {attribute 'hide'}
    bDelayReadAtInit 		 : BOOL;
    bBaseExec: BOOL;
    nCommandLocal  			 : E_MCS2OpMode := E_MCS2OpMode.CSP;
END_VAR

VAR CONSTANT
    {attribute 'hide'}
    nChanSoftLimitBase       : WORD := 16#200E;
    {attribute 'hide'}
    nChanHomeOffsetBase      : WORD := 16#607C;
    {attribute 'hide'}
    nChanHomeMethodBase      : WORD := 16#6098;
    {attribute 'hide'}
    nChanHomingSpeedBase     : WORD := 16#6099;
    {attribute 'hide'}
    nChanhomingAccBase       : WORD := 16#609A;
    {attribute 'hide'}
    nChanErrorCodeBase       : WORD := 16#603F;
    {attribute 'hide'}
    nChanFErrWinBase         : WORD := 16#6065;
    {attribute 'hide'}
    nChanOfsBase             : WORD := 16#800;      // For SmartAct MCS2 and E-727
    {attribute 'hide'}
    nChanEncErrorCode        : WORD := 16#7300;     // Motor encoder defective code (for save/restore)
    {attribute 'hide'}
    nChanSoftLimBase         : WORD := 16#200E;
    {attribute 'hide'}
    nChanOlStepBase          : WORD := 16#2022;
    {attribute 'hide'}
    nChanOlStepAmpBase       : WORD := 16#2023;
    {attribute 'hide'}
    nChanOlStepFreqBase      : WORD := 16#2024;
    {attribute 'hide'}
    nChanMaxCloseLoopFreqBase: WORD := 16#2001;
    {attribute 'hide'}
    nChanPositionerTypeBase  : WORD := 16#2000;
    {attribute 'hide'}
    nCHanCalibrationOptBase  : WORD := 16#2004;
    {attribute 'hide'}
    nChanSensorPowerModeBase : WORD := 16#2007;
    {attribute 'hide'}
    nChanReferencingOptBase  : WORD := 16#200B;
    {attribute 'hide'}
    nChanReferenceTypeBase   : WORD := 16#200A;
    {attribute 'hide'}
    nChanSafeDirBase         : WORD := 16#200C;
    {attribute 'hide'}
    nChanMotorLoadBase       : WORD := 16#200D;
    {attribute 'hide'}
    nChannelTypeBase         : WORD := 16#200F;
    {attribute 'hide'}
    nChannelStateBase        : WORD := 16#2025;
    {attribute 'hide'}
    nChanLogicalScaleOffsetBase  : WORD := 16#2008;
    {attribute 'hide'}
    nChanLogicalScaleInvBase     : WORD := 16#2009;
    {attribute 'hide'}
    nChanChannelTempBase         : WORD := 16#2026;
    {attribute 'hide'}
    nChanMovementTypeBase        : WORD := 16#2003;
    {attribute 'hide'}
    nChanBaseUnitBase            : WORD := 16#2005;
    {attribute 'hide'}
    nChanBaseResolutionBase      : WORD := 16#2006;
    {attribute 'hide'}
    nChanDistCodeInvBase         : WORD := 16#2029;
    {attribute 'hide'}
    nChanPositionerCtrlOptBase   : WORD := 16#2027;
    {attribute 'hide'}
    nChanActuatorModeBase        : WORD := 16#2028;
    {attribute 'hide'}
    nChanMotorLoadProtBase       : WORD := 16#202B;
    {attribute 'hide'}
    nChanDiagClfBase             : WORD := 16#202A;
    // Held as constants so the retract check below cannot drift from the text posted.
    {attribute 'hide'}
    sMsgPosLimit                 : STRING := 'Cannot move past positive limit.';
    {attribute 'hide'}
    sMsgNegLimit                 : STRING := 'Cannot move past Negative limit.';
END_VAR

VAR PERSISTENT
    bSaved                   : BOOL;
    fSavedPosition           : LREAL;
    bLastPositiveDirection   : BOOL;
    bLastNegativeDirection   : BOOL;
END_VAR

IF NOT __ISVALIDREF(stMotionStage)
OR NOT __ISVALIDREF(stChanParams) THEN
    RETURN;
END_IF

// When the PLC autoboots, I/O is not yet valid after 'call_after_init'
IF bSystemInit THEN
    IF stMotionStage.Axis.NcToPlc.AxisId <> 0 THEN
        bExecParamRead	:= TRUE;
        stChanParams.bStageReady  := TRUE;
        bSystemInit	:= FALSE;
        stChanParams.fPosition    := stMotionStage.Axis.NcToPlc.ActPos;
    END_IF
END_IF

(*
  Shortcut command edge detection
  Move requests can arrive via bMoveCmd (shortcut) or directly via bExecute
*)
rtMoveCmdShortcut    (CLK := stMotionStage.bMoveCmd);
rtHomeCmdShortcut    (CLK := stMotionStage.bHomeCmd);
rtStepCmdShortcut    (CLK := stChanParams.bStepMoveCmd);
rtStepFwdCmdShortcut (CLK := stChanParams.bStepForwardCmd);
rtStepRevCmdShortcut (CLK := stChanParams.bStepReverseCmd);
rtCalibrateCmdShortcut(CLK := stChanParams.bCalibrationCmd);

IF rtMoveCmdShortcut.Q AND NOT stMotionStage.bExecute THEN
    stMotionStage.bExecute := TRUE;
    stMotionStage.nCommand := E_EpicsMotorCmd.MOVE_ABSOLUTE;
    bEnPosLag              := bRecentEnPosLagStatus;
    fParameterValue        := BOOL_TO_LREAL(bRecentEnPosLagStatus);

ELSIF rtStepCmdShortcut.Q AND NOT stMotionStage.bExecute THEN
    stMotionStage.bExecute := TRUE;
    stMotionStage.nCommand := E_EpicsMotorCmd.JOG;
    bEnPosLag              := bRecentEnPosLagStatus;
    fParameterValue        := BOOL_TO_LREAL(bRecentEnPosLagStatus);

ELSIF rtStepFwdCmdShortcut.Q AND NOT stMotionStage.bExecute THEN
    // Forward jog: drive the step count positive, then step
    stChanParams.nChanStep := ABS(stChanParams.nChanStep);
    stMotionStage.bExecute := TRUE;
    stMotionStage.nCommand := E_EpicsMotorCmd.JOG;
    bEnPosLag              := bRecentEnPosLagStatus;
    fParameterValue        := BOOL_TO_LREAL(bRecentEnPosLagStatus);

ELSIF rtStepRevCmdShortcut.Q AND NOT stMotionStage.bExecute THEN
    // Reverse jog: drive the step count negative, then step
    stChanParams.nChanStep := -ABS(stChanParams.nChanStep);
    stMotionStage.bExecute := TRUE;
    stMotionStage.nCommand := E_EpicsMotorCmd.JOG;
    bEnPosLag              := bRecentEnPosLagStatus;
    fParameterValue        := BOOL_TO_LREAL(bRecentEnPosLagStatus);

ELSIF rtCalibrateCmdShortcut.Q AND NOT stMotionStage.bExecute THEN
    stMotionStage.bExecute := TRUE;
    stMotionStage.nCommand := E_EpicsMotorCmd.CALIBRATE;
    bRecentEnPosLagStatus := stMotionStage.stAxisParameters.bCtrlEnablePosDiffControl.0;
    // Trigger WriteParameterNC to disable position lag during calibration.
    bEnPosLag             := bRecentEnPosLagStatus;
    // Write 0 = disable position lag monitoring.
    fParameterValue       := 0;
    bLagClearPending      := bRecentEnPosLagStatus;

ELSIF rtHomeCmdShortcut.Q AND NOT stMotionStage.bExecute THEN
    stMotionStage.nCommand := E_EpicsMotorCmd.HOME;
    stMotionStage.nCmdData := stChanParams.eHomeMode;
    stMotionStage.bExecute := (stChanParams.eHomeMode = E_MCS2HomeMethod.AutoMethod)
                              OR (stChanParams.eHomeMode = E_MCS2HomeMethod.CurrentPositionMethod);

    bRecentEnPosLagStatus := stMotionStage.stAxisParameters.bCtrlEnablePosDiffControl.0;
    // Trigger WriteParameterNC to disable position lag during homing.
    bEnPosLag             := bRecentEnPosLagStatus;
    // Write 0 = disable position lag monitoring.
    fParameterValue       := 0;
    bLagClearPending      := bRecentEnPosLagStatus;
END_IF

// Main execute edge: covers both shortcut and direct bExecute paths
rtUserExec(CLK := stMotionStage.bExecute);

// Valid move request: not busy, rising execute edge, no error
bNewMoveReq S= NOT stMotionStage.bBusy AND rtUserExec.Q AND NOT stMotionStage.bError;
bNewMoveReq R= NOT stMotionStage.bExecute OR stMotionStage.bError;
bPrepareDisable R= bNewMoveReq;

IF rtUserExec.Q THEN
    //nCommandLocal := stMotionStage.nCommand;
    // Cover direct bExecute path, shortcut path already set bEnPosLag/fParameterValue
    IF NOT rtMoveCmdShortcut.Q
        AND NOT rtStepCmdShortcut.Q
        AND NOT rtCalibrateCmdShortcut.Q
        AND NOT rtHomeCmdShortcut.Q
    THEN
        IF stMotionStage.nCommand = E_EpicsMotorCmd.HOME
            OR stMotionStage.nCommand = E_EpicsMotorCmd.CALIBRATE THEN
            bRecentEnPosLagStatus := stMotionStage.stAxisParameters.bCtrlEnablePosDiffControl.0;
            bEnPosLag             := bRecentEnPosLagStatus;
            fParameterValue       := 0;
            bLagClearPending      := bRecentEnPosLagStatus;
        ELSE
            bEnPosLag       := bRecentEnPosLagStatus;
            fParameterValue := BOOL_TO_LREAL(bRecentEnPosLagStatus);
        END_IF
    END_IF

    IF NOT stMotionStage.bHomeCmd
        AND NOT stChanParams.stChannelState.bIsReferenced THEN
        IF stChanParams.eHomeMode <> E_EpicsHomeCmd.NONE
            AND NOT stMotionStage.bHomed THEN
            stMotionStage.sErrorMessage := 'Axis homing mode set, but homing routine pending';
        END_IF
    END_IF
END_IF

// Drive manager
fbDriveManager(
    stMotionStage        := stMotionStage,
    stDS402Drive         := stDS402Drive,
    stMCS2ChanParameter  := stChanParams,
    bUserExec            := rtUserExec.Q,
    eRequestedManualMode => nCommandLocal
);

// Enable mode handling
rtEnableMode(CLK := (stMotionStage.nEnableMode = E_StageEnableMode.DURING_MOTION));

CASE stMotionStage.nEnableMode OF
    E_StageEnableMode.ALWAYS:
        stMotionStage.bEnable := stMotionStage.bSafetyReady;

    E_StageEnableMode.DURING_MOTION:
        IF rtEnableMode.Q THEN
            stMotionStage.bEnable := FALSE;
        END_IF
        IF bNewMoveReq THEN
            bPositionHold        := FALSE;
            tonHoldTime.IN       := FALSE;
            stMotionStage.bEnable:= stMotionStage.bSafetyReady;
            bLastHoltTimeOut     := FALSE;
            bHalt                := FALSE;
        END_IF
END_CASE

// Interlock: Reacts on internal limit conditions
Interlock();

bBaseExec := NOT stMotionStage.bError
             AND stMotionStage.bExecute
             AND stMotionStage.bAllEnable
             AND stMotionStage.bSafetyReady;

IF fbDriveManager.bCSPModeEnabled THEN
    // Close loop: gate on NC standstill state (bEnableDone)
    bLocalExec := bBaseExec
                  AND stMotionStage.bEnableDone
                  AND stMotionStage.nCommand = E_EpicsMotorCmd.MOVE_ABSOLUTE;

ELSIF fbDriveManager.bHomeModeEnabled THEN
    // Open loop homing: gate on DS402 operational state
    bLocalExec := bBaseExec
                  AND fbDriveManager.bOperational
                  AND stMotionStage.nCommand = E_EpicsMotorCmd.HOME;

ELSIF fbDriveManager.bStepModeEnabled THEN
    // Open loop step: gate on DS402 operational state
    bLocalExec := bBaseExec
                  AND fbDriveManager.bOperational
                  AND stMotionStage.nCommand = E_EpicsMotorCmd.JOG;

ELSIF fbDriveManager.bCalibrationModeEnabled THEN
    // Open loop calibration: gate on DS402 operational state
    bLocalExec := bBaseExec
                  AND fbDriveManager.bOperational
                  AND stMotionStage.nCommand = E_EpicsMotorCmd.CALIBRATE;
ELSE
    bLocalExec := FALSE;
END_IF

bExecMove := bLocalExec AND ((stMotionStage.nCommand = E_EpicsMotorCmd.MOVE_ABSOLUTE)
                          OR  (stMotionStage.nCommand = E_EpicsMotorCmd.JOG)
                          OR  (stMotionStage.nCommand = E_EpicsMotorCmd.CALIBRATE));
bExecHome := bLocalExec AND NOT bExecMove;

rtExec(CLK := bLocalExec);
IF rtExec.Q THEN
    stDS402Drive.nDriveControl.8 := FALSE;
    stMotionStage.bDone          := FALSE;
END_IF


IF NOT fbDriveManager.bDS402Manual THEN
    stMotionStage.Axis.ReadStatus();
END_IF

// Get definitive bEnableDone from NC axis state
CASE stMotionStage.Axis.Status.MotionState OF
    MC_AXISSTATE_UNDEFINED, MC_AXISSTATE_DISABLED, MC_AXISSTATE_ERRORSTOP:
        stMotionStage.bEnableDone := FALSE;
    ELSE
        stMotionStage.bEnableDone := TRUE;
END_CASE

// Reset handling
IF stMotionStage.bReset THEN
    stMotionStage.bExecute          := FALSE;
    stMotionStage.bError            := FALSE;
    stMotionStage.nErrorId          := 0;
    stMotionStage.sErrorMessage     := '';
    stMotionStage.sCustomErrorMessage := '';
    stChanParams.nMCS2ErrorCode     := 0;
    stChanParams.sMCS2ErrorMessage   := '';
    fbStepMode.Reset();
    fbhome.Reset();
    bReset := TRUE;
    bLagClearPending := FALSE;
    IF fbDriveManager.bDS402Manual THEN
        stDS402Drive.nDriveControl.7 := TRUE;
    END_IF
    stMotionStage.bReset := FALSE;
END_IF

// Stop/halt detection. bHalt is the user-stop channel only: execute dropped
// mid-move. Limit reaction is handled by the direction enables, not from here.
ftExec(CLK := stMotionStage.bExecute);
bHalt := ftExec.Q AND stMotionStage.bBusy;
rtHaltEdge(CLK := bHalt);
IF rtHaltEdge.Q AND fbDriveManager.bDS402Manual THEN
    fbStepMode.Halt();
    fbhome.Halt();
    stDS402Drive.nDriveControl.8 := TRUE;
END_IF

WriteParameterNC(
    Execute         := bEnPosLag,
    ParameterNumber := MC_AxisParameter.AxisEnPositionLagMonitoring,
    ParameterValue  := fParameterValue
);

// Hold the open-loop home/calibrate move until the NC position-lag disable actually
// lands, so the drive's referencing move cannot trip a following error on residual lag
// monitoring. Timeout caps the wait so a missing write cannot hang the routine.
rtMcWriteDone(CLK := fbMcWriteParameter.Done);
tonLagClearTimeout(IN := bLagClearPending, PT := T#500MS);
IF bLagClearPending
   AND ((fParameterValue = 0 AND rtMcWriteDone.Q) OR tonLagClearTimeout.Q) THEN
    bLagClearPending := FALSE;
END_IF

bParamsEnable := stMotionStage.bAxisParamsInit AND stChanParams.bEnableHardwareOps;

fbWriteParameters(
    bEnable             := bParamsEnable,
    bErrorAcknowledge   := stMotionStage.bReset,
    stDS402Drive        := stDS402Drive,
    stMotionStage       := stMotionStage,
    stChanParams := stChanParams
);

CASE nCommandLocal OF
    E_MCS2OpMode.CSP:
        Reset();
        Power();
        Halt();
        (*Wait for drive to be in the correct mode after a request was validated *)
        MoveAbsolute();
        (*
          IN CSP mode the drive control word is update via the NC
          Manual step mode and Homing will override this
        *)

        stDS402Drive.nModeOfOperation := stDS402Drive.nModeOfOperationNC;
        stDS402Drive.nDriveControl    := stDS402Drive.nDriveControlNC;

    E_MCS2OpMode.HOME:
        (*DS402 Manual Homing*)
        // Gate on the drive manager confirming HOME mode is active and operational.
        fbhome(
            bExecute := bExecHome AND fbWriteParameters.bParamsSet AND NOT bLagClearPending
                        AND fbDriveManager.bHomeModeEnabled,
            stDS402Drive  := stDS402Drive,
            stMotionStage := stMotionStage
        );

    E_MCS2OpMode.STEP:
        fbStepMode(
            bExecute       := bExecMove AND fbWriteParameters.bParamsSet
                              AND fbDriveManager.bStepModeEnabled,
            stDS402Drive  := stDS402Drive,
            stMotionStage := stMotionStage
        );

    E_MCS2OpMode.CALIBRATE:
        fbCalibrate(
            bExecute	 := bExecMove AND fbWriteParameters.bParamsSet AND NOT bLagClearPending
                          AND fbDriveManager.bCalibrationModeEnabled,
            stDS402Drive  := stDS402Drive,
            stMotionStage := stMotionStage
        );
END_CASE

stMotionStage.bBusy := fbMcMoveAbsolute.Busy
                       OR fbhome.bHomeMoveBusy
                       OR fbStepMode.bStepMoveBusy
                       OR fbCalibrate.bCalibrateMoveBusy;
// Check done moving via user stop, limit hit, Target Position reached, or from homing.
PostMoveChecks();
// update encoder value and calibrated position
ScaleEncRawValue();
// Drive parameters
ExposedParameters(Enable := stChanParams.bStageReady, tRefreshDelay := T#2S);
// Read MCS2 Channel Parameters
fbReadChanParams(
    bEnable             := bParamsEnable,
    stMotionStage       := stMotionStage,
    stMCS2ChanParameter := stChanParams,
    stDS402Drive        := stDS402Drive,
);
(* Save and restore as long as not an absolute encoder*)
PersistParameters(Enable := stChanParams.bStageReady);
(*Restore encoder value at initialization*)
RestoreMotionParams(Enable := stChanParams.bStageReady);
(*EPICS Motor record Update*)
UpdateEpicsStatus();

(*
    Error from functions and Nc. The error will send to EPICS interface based on predifined
    priority: axis, power, backlash, absoluteMove, etc...
*)
IF fbMcPower.Error AND fbMcPower.Active THEN
    stMotionStage.bError   := fbMcPower.Error;
    stMotionStage.nErrorId := fbMcPower.ErrorID;
ELSIF fbMcMoveAbsolute.Error THEN
    stMotionStage.bError   := fbMcMoveAbsolute.Error;
    stMotionStage.nErrorId := fbMcMoveAbsolute.ErrorID;
ELSIF fbMcHalt.Error AND fbMcHalt.Active THEN
    stMotionStage.bError   := fbMcHalt.Error;
    stMotionStage.nErrorId := fbMcHalt.ErrorID;
ELSIF fbMcReset.Error THEN
    stMotionStage.bError   := fbMcReset.Error;
    stMotionStage.nErrorId := fbMcReset.ErrorID;
ELSIF fbMcWriteParameter.Error THEN
    stMotionStage.bError   := fbMcWriteParameter.Error;
    stMotionStage.nErrorId := fbMcWriteParameter.ErrorID;
ELSIF fbMcReadParams.Error AND NOT stMotionStage.bBusy THEN
    stMotionStage.bError   := fbMcReadParams.Error;
    stMotionStage.nErrorId := fbMcReadParams.ErrorID;
ELSE
    IF stMotionStage.bBusy THEN
        // Clear the display message during normal motion, but leave sCustomErrorMessage
        // intact: Interlock may have just set it on this same cycle, and the NC error
        // that latches bError will not be visible until the next cycle.
        stMotionStage.sErrorMessage := '';
    END_IF
END_IF

(*Double function, prioritize NC error otherwise read drive channel error code*)
fbReadDriveCodes(
    bEnable             := bParamsEnable,
    stMotionStage       := stMotionStage,
    stMCS2ChanParameter := stChanParams,
    stDS402Drive        := stDS402Drive,
);

IF stMotionStage.sCustomErrorMessage <> ''
    AND stMotionStage.sErrorMessage = '' THEN
    stMotionStage.sErrorMessage := stMotionStage.sCustomErrorMessage;
END_IF

(*Clear motion flag when error occurs*)
IF stMotionStage.bError THEN
    stMotionStage.bExecute := FALSE;
    stMotionStage.bBusy    := FALSE;
    stMotionStage.bDone    := FALSE;
    stMotionStage.bEnable  := FALSE;
END_IF

(* We've got the rising edge clear these flags.*)
stMotionStage.bMoveCmd             := FALSE;
stMotionStage.bHomeCmd             := FALSE;
stChanParams.bStepMoveCmd   := FALSE;
stChanParams.bStepForwardCmd := FALSE;
stChanParams.bStepReverseCmd := FALSE;
stChanParams.bCalibrationCmd := FALSE;

METHOD PUBLIC  ExposedParameters
VAR_INPUT
    Enable : BOOL;
    tRefreshDelay: TIME;
END_VAR

VAR_INST
    {attribute 'hide'}
    bParamReadTimer     : BOOL := TRUE;
END_VAR
// Periodic update of NC parameters
NCParamsTimer( IN:=Enable AND NOT bExecParamRead, PT:=tRefreshDelay);
bExecParamRead S= NCParamsTimer.Q;
fbMcReadParams(
    Parameter:= stMotionStage.stAxisParameters,
    Axis:= stMotionStage.Axis,
    Execute:= bExecParamRead );

// Copy axis parameters that we want to expose to the EPICS layer.
 stMotionStage.stAxisParametersExposed.bCtrlEnablePosDiffControl     :=  stMotionStage.stAxisParameters.bCtrlEnablePosDiffControl;
 stMotionStage.stAxisParametersExposed.bEncEnableSoftEndMaxControl   :=  stMotionStage.stAxisParameters.bEncEnableSoftEndMaxControl;
 stMotionStage.stAxisParametersExposed.bEncEnableSoftEndMinControl   :=  stMotionStage.stAxisParameters.bEncEnableSoftEndMinControl;
 stMotionStage.stAxisParametersExposed.fAccelerationMax              :=  stMotionStage.stAxisParameters.fAccelerationMax;
 stMotionStage.stAxisParametersExposed.fCtrlPosDiffMax               :=  stMotionStage.stAxisParameters.fCtrlPosDiffMax;
 stMotionStage.stAxisParametersExposed.fCtrlPosDiffMaxTime           :=  stMotionStage.stAxisParameters.fCtrlPosDiffMaxTime;
 stMotionStage.stAxisParametersExposed.fDecelerationMax              :=  stMotionStage.stAxisParameters.fDecelerationMax;
 stMotionStage.stAxisParametersExposed.fEncSoftEndMax                :=  stMotionStage.stAxisParameters.fEncSoftEndMax;
 stMotionStage.stAxisParametersExposed.fEncSoftEndMin                :=  stMotionStage.stAxisParameters.fEncSoftEndMin;
 stMotionStage.stAxisParametersExposed.fVeloMaximum                  :=  stMotionStage.stAxisParameters.fVeloMaximum;
 stMotionStage.stAxisParametersExposed.fEncOffset                       :=  stMotionStage.stAxisParameters.fEncOffset;
 stMotionStage.stAxisParametersExposed.fEncScaleFactorInternal       :=  stMotionStage.stAxisParameters.fEncScaleFactorInternal;

bExecParamRead R= fbMcReadParams.Done OR fbMcReadParams.Error;
 stMotionStage.bAxisParamsInit S= fbMcReadParams.Done;
END_METHOD

//FB_Init is always available implicitly and it is used primarily for initialization.
//The return value is not evaluated. For a specific influence, you can also declare the
//methods explicitly and provide additional code there with the standard initialization
//code. You can evaluate the return value.
METHOD FB_Init: BOOL
VAR_INPUT
    bInitRetains: BOOL; // TRUE: the retain variables are initialized (reset warm / reset cold)
    bInCopyCode: BOOL;  // TRUE: the instance will be copied to the copy code afterward (online change)
    stMotionStage	: REFERENCE TO ST_MotionStage;
    stMCS2ChanParameter : REFERENCE TO ST_MCS2ChanParameter;
    (*Mandatory must be unique for each MCS2 axis *)
    eModule : E_Module;
END_VAR
THIS^.stMotionStage REF= stMotionStage;
THIS^.stChanParams REF= stMCS2ChanParameter;
THIS^.eModule := eModule;
END_METHOD

METHOD Halt
fbMcHalt(
    Axis :=  stMotionStage.Axis,
    Execute := bHalt,
    Deceleration :=  stMotionStage.fDeceleration,
    BufferMode := MC_BufferMode.MC_Aborting,
);
IF fbMcHalt.Done THEN
    bHalt := FALSE;
END_IF
END_METHOD

METHOD PUBLIC Interlock

VAR_INST
    {attribute 'hide'}
    bPositiveDirection  : BOOL;
    {attribute 'hide'}
    bNegativeDirection  : BOOL;
    {attribute 'hide'}
    ftForwardEnabled    : F_TRIG;
    {attribute 'hide'}
    ftBackwardEnabled   : F_TRIG;
    {attribute 'hide'}
    bHitForwardLimit    : BOOL;
    {attribute 'hide'}
    bHitBackwardLimit   : BOOL;
    {attribute 'hide'}
    fCurrentPosition    : LREAL;
END_VAR
// Positive or Negative direction.
// In step mode fPosDiff is unreliable for direction: fPosition is the stale NC setpoint
// and fMeasuredPos is the live encoder, so their difference inverts as the motor moves.
// Use the step count sign instead, which is set explicitly at command issue time.
IF fbDriveManager.bStepModeEnabled THEN
    bPositiveDirection := stMotionStage.bBusy AND stChanParams.nChanStep > 0;
    bNegativeDirection := stMotionStage.bBusy AND stChanParams.nChanStep < 0;
ELSE
    bPositiveDirection := stMotionStage.bBusy AND stMotionStage.fPosDiff > 0;
    bNegativeDirection := stMotionStage.bBusy AND stMotionStage.fPosDiff < 0;
END_IF

// If the drive starts limited and no direction history is available, infer the
// blocked side from the nearest configured software range limit. The aggregate
// InternalLimitActive bit does not identify the side by itself.
fCurrentPosition := DINT_TO_LREAL(stMotionStage.nRawEncoderDINT)
                    * MAX(stMotionStage.stAxisParameters.fEncScaleFactorInternal,
                          stChanParams.fScalingFactor);
IF stDS402Drive.stDriveStatus.InternalLimitActive THEN
    IF NOT bLastPositiveDirection AND NOT bLastNegativeDirection THEN
        IF fbReadChanParams.bAllReadsComplete THEN
            IF stChanParams.nSoftLimMax > stChanParams.nSoftLimMin THEN
                IF ABS(fCurrentPosition - stChanParams.nSoftLimMin)
                   < ABS(stChanParams.nSoftLimMax - fCurrentPosition) THEN
                    bLastNegativeDirection := TRUE;
                ELSE
                    bLastPositiveDirection := TRUE;
                END_IF
            END_IF
        END_IF
    END_IF
END_IF

// Preserve the last commanded direction across the stop and PLC restart. The
// drive exposes one aggregate limit bit, so this retained context identifies
// which direction should remain blocked during recovery.
IF NOT stDS402Drive.stDriveStatus.InternalLimitActive
    OR (NOT bHitForwardLimit AND NOT bHitBackwardLimit) THEN
    IF bPositiveDirection THEN
        bLastPositiveDirection := TRUE;
        bLastNegativeDirection := FALSE;
    ELSIF bNegativeDirection THEN
        bLastPositiveDirection := FALSE;
        bLastNegativeDirection := TRUE;
    END_IF
END_IF

// Latch which physical limit was hit; clear once the drive is no longer reporting a limit.
// A single InternalLimitActive bit covers both directions, so direction at the time of
// the hit is used to determine which enable to hold off.
bHitForwardLimit  S= stDS402Drive.stDriveStatus.InternalLimitActive
                   AND (bPositiveDirection OR bLastPositiveDirection);
bHitBackwardLimit S= stDS402Drive.stDriveStatus.InternalLimitActive
                    AND (bNegativeDirection OR bLastNegativeDirection);
bHitForwardLimit  R= NOT stDS402Drive.stDriveStatus.InternalLimitActive;
bHitBackwardLimit R= NOT stDS402Drive.stDriveStatus.InternalLimitActive;

// An active limit with no known direction disables both directions. Once the
// hit direction is known, only that direction is disabled for reverse recovery.
stMotionStage.bLimitForwardEnable := NOT stDS402Drive.stDriveStatus.InternalLimitActive
                                     OR (bHitBackwardLimit AND NOT bHitForwardLimit);
stMotionStage.bLimitBackwardEnable := NOT stDS402Drive.stDriveStatus.InternalLimitActive
                                      OR (bHitForwardLimit AND NOT bHitBackwardLimit);

// use falling trigger to avoid spamming sErrorMessage
ftForwardEnabled(CLK := stMotionStage.bLimitForwardEnable);
ftBackwardEnabled(CLK := stMotionStage.bLimitBackwardEnable);

// A limit hit is the lowest priority message. Never post one over a latched fault,
// and retract our own once the drive releases the limit so a stale warning cannot
// later be promoted into sErrorMessage. The drive stops the positioner itself and
// SetEnables drops the offending direction, so no halt is requested here.
IF NOT stMotionStage.bError AND NOT fbhome.bHomeMoveBusy THEN
    IF bHitForwardLimit AND ftForwardEnabled.Q THEN
        stMotionStage.sCustomErrorMessage := sMsgPosLimit;
    ELSIF bHitBackwardLimit AND ftBackwardEnabled.Q THEN
        stMotionStage.sCustomErrorMessage := sMsgNegLimit;
    END_IF
END_IF

IF NOT bHitForwardLimit AND NOT bHitBackwardLimit
   AND (stMotionStage.sCustomErrorMessage = sMsgPosLimit
        OR stMotionStage.sCustomErrorMessage = sMsgNegLimit) THEN
    stMotionStage.sCustomErrorMessage := '';
END_IF

IF NOT  stMotionStage.bError AND  stMotionStage.bExecute AND NOT  stMotionStage.bUserEnable THEN
     stMotionStage.bError := TRUE;
     stMotionStage.nErrorId := 1;
     stMotionStage.sCustomErrorMessage := 'Move requested, but user enable is disabled!';
END_IF

// Update all enable booleans
SetEnables();
END_METHOD

METHOD PUBLIC  MoveAbsolute
fbMcMoveAbsolute(
    Axis :=  stMotionStage.Axis,
    Execute := bExecMove AND fbMcPower.Status AND fbDriveManager.bCSPModeEnabled,
    Position :=  stMotionStage.fPosition,
    Velocity :=  stMotionStage.fVelocity,
    Acceleration :=  stMotionStage.fAcceleration,
    Deceleration :=  stMotionStage.fDeceleration,
    BufferMode := MC_BufferMode.MC_Aborting,
);

IF fbMcMoveAbsolute.Done (*OR fbMcReset.Done*) THEN
    (*Hold the position in close loop before dropping power, a positional drift will occur then*)
    IF ( stMotionStage.nEnableMode = E_StageEnableMode.DURING_MOTION ) THEN
        bPositionHold := TRUE;
        tonHoldTime.IN:=TRUE;
    END_IF
END_IF
END_METHOD

METHOD PersistParameters
VAR_INPUT
    Enable  : BOOL;
END_VAR

